    // Проверка правил
    FOR L_j := 1 TO GVL_CONSTANTS.C_MAX_RULES DO
        IF VI_Rule_Actions[L_j].Active AND VI_Rule_Actions[L_j].Target_ID = L_i THEN
            IF VI_Rule_Actions[L_j].Action_Type = E_Rule_Action_Type.ACTION_SET_LIGHTING_BASE THEN
                L_Rule_Light_Active := TRUE;
                L_Rule_Light_Val := REAL_TO_BYTE(VI_Rule_Actions[L_j].Value);
                L_Light_States[L_i] := (L_Rule_Light_Val > 0);
            ELSIF VI_Rule_Actions[L_j].Action_Type = E_Rule_Action_Type.ACTION_TOGGLE_LIGHTING AND VI_Rule_Actions[L_j].Triggered THEN
                L_Light_States[L_i] := NOT L_Light_States[L_i];
            END_IF;
        END_IF;
    END_FOR;

    // Приоритет 1: Физические выключатели (ТЗ 1.0)
    IF VI_Physical_Switches[L_i] AND NOT L_Prev_Switches[L_i] THEN
        L_Light_States[L_i] := NOT L_Light_States[L_i];
        L_Manual_Override[L_i] := TRUE; // Запоминаем ручное переопределение
    END_IF;
    L_Prev_Switches[L_i] := VI_Physical_Switches[L_i];

    // Приоритет 2: Датчики движения (ТЗ 2.0)
    // Защита от дребезга и удержание сигнала движения с помощью TOF
    L_Motion_Timers[L_i](IN := VI_Motion_Sensors[L_i], PT := T#5m, VI_System_Time_MS := VI_System_Time_MS);
    
    // Сброс ручного переопределения, когда комната становится пустой (задний фронт таймера движения)
    IF L_Prev_Motion_Q[L_i] AND NOT L_Motion_Timers[L_i].Q THEN
        L_Manual_Override[L_i] := FALSE;
    END_IF;
    L_Prev_Motion_Q[L_i] := L_Motion_Timers[L_i].Q;

    IF L_Motion_Timers[L_i].Q THEN
        IF NOT L_Manual_Override[L_i] THEN
            L_Light_States[L_i] := TRUE;
        END_IF;
    ELSE
        // Выключаем свет только если нет ручного переопределения
        IF NOT L_Manual_Override[L_i] THEN
            L_Light_States[L_i] := FALSE;
        END_IF;
    END_IF;

    // Приоритет 3: Симуляция (только в режиме Away)
    IF L_Effective_Scenario = E_SCENARIO_TYPE.SCENARIO_AWAY AND L_Effective_Simulation_Active THEN
        L_Light_States[L_i] := VI_Simulation_Lights[L_i];
    END_IF;

    // Приоритет 4: Ручное управление и правила
    IF VI_Manual_Light_Override[L_i] > 0 THEN
        VO_Lighting_Levels[L_i] := VI_Manual_Light_Override[L_i];
    ELSIF L_Rule_Light_Active THEN
        VO_Lighting_Levels[L_i] := L_Rule_Light_Val;
    ELSE
        VO_Lighting_Levels[L_i] := SEL(L_Light_States[L_i], 0, L_Base_Light);
    END_IF;
    
    // 5. Мокрые зоны
    IF VI_Wet_Zone_Map[L_i] AND L_Wet_Zone_Idx <= GVL_CONSTANTS.C_MAX_WET_ZONES THEN
        VO_Wet_Zone_Light_Active[L_Wet_Zone_Idx] := (VO_Lighting_Levels[L_i] > 10);
        L_Wet_Zone_Idx := L_Wet_Zone_Idx + 1;
    END_IF;
END_FOR;

// 3. Управление шторами
FOR L_i := 1 TO GVL_CONSTANTS.C_MAX_BLINDS DO
    L_Rule_Blinds_Active := FALSE;
    L_Rule_Blinds_Val := 0;
    
    // Проверка правил
    FOR L_j := 1 TO GVL_CONSTANTS.C_MAX_RULES DO
        IF VI_Rule_Actions[L_j].Active AND VI_Rule_Actions[L_j].Target_ID = L_i THEN
            IF VI_Rule_Actions[L_j].Action_Type = E_Rule_Action_Type.ACTION_SET_BLINDS THEN
                L_Rule_Blinds_Active := TRUE;
                L_Rule_Blinds_Val := REAL_TO_BYTE(VI_Rule_Actions[L_j].Value);
            END_IF;
        END_IF;
    END_FOR;

    // Приоритет 1: Ручное управление
    IF VI_Manual_Blinds_Override[L_i] > 0 THEN
        VO_Blinds_Positions[L_i] := VI_Manual_Blinds_Override[L_i];
    // Приоритет 2: Правила
    ELSIF L_Rule_Blinds_Active THEN
        VO_Blinds_Positions[L_i] := L_Rule_Blinds_Val;
    // Приоритет 3: Сценарий
    ELSE
        VO_Blinds_Positions[L_i] := L_Base_Blinds;
    END_IF;
END_FOR;

// ========================================
// Lighting V2 shadow execution (phase2)
// ========================================
fbLightingV2Staging(
    VI_Zone_ID := 1,
    VI_Enable := (VO_Lighting_Levels[1] > 0),
    VI_Brightness_Setpoint := BYTE_TO_REAL(VO_Lighting_Levels[1]),
    VI_Scene_ID := TO_INT(L_Effective_Scenario),
    VI_Manual_Override := (VI_Manual_Light_Override[1] > 0),
    VI_Transition_Time_MS := 5000,

    VI_Is_Active := (VO_Lighting_Levels[1] > 0),
    VI_Brightness_Actual := BYTE_TO_REAL(VO_Lighting_Levels[1]),
    VI_Motion_Active := VI_Motion_Sensors[1],
    VI_Ambient_Lux := 0.0,
    VI_Alarm_Active := GVL_STATE.G_Lighting_IO_Fault OR GVL_STATE.G_Lighting_Subsystem_Degraded,

    VO_Command_Shadow => L_Lighting_V2_Command_Shadow,
    VO_State_Shadow => L_Lighting_V2_State_Shadow
);

// ========================================
// Lighting V2 shadow validation
// ========================================
IF ABS(BYTE_TO_REAL(VO_Lighting_Levels[1]) - L_Lighting_V2_Command_Shadow.Brightness_Setpoint) > 0.1 THEN
    L_Lighting_V2_Shadow_Diff_Found := TRUE;
END_IF;
IF ABS(BYTE_TO_REAL(VO_Lighting_Levels[1]) - L_Lighting_V2_State_Shadow.Brightness_Actual) > 0.1 THEN
    L_Lighting_V2_Shadow_Diff_Found := TRUE;
END_IF;
IF VI_Motion_Sensors[1] <> L_Lighting_V2_State_Shadow.Motion_Active THEN
    L_Lighting_V2_Shadow_Diff_Found := TRUE;
END_IF;

// Guarded Lighting V2 enable
IF L_Lighting_V2_Switch_Enabled THEN
    IF NOT L_Lighting_V2_Shadow_Diff_Found THEN
        L_Lighting_V2_Path_Ready := TRUE;
        L_Lighting_Using_Legacy_Fallback := FALSE;
    ELSE
        L_Lighting_V2_Path_Ready := FALSE;
        L_Lighting_Using_Legacy_Fallback := TRUE;
    END_IF;
ELSE
    L_Lighting_V2_Path_Ready := FALSE;
    L_Lighting_Using_Legacy_Fallback := TRUE;
END_IF;



// ========================================
// Blinds V2 shadow execution (phase2)
// ========================================
fbBlindsV2Staging(
    VI_Blind_ID := 1,
    VI_Enable := TRUE,
    VI_Position_Setpoint := VO_Blinds_Positions[1],
    VI_Manual_Override := (VI_Manual_Blinds_Override[1] > 0),
    VI_Scenario_ID := TO_INT(L_Effective_Scenario),
    VI_Safety_Mode := FALSE,

    VI_Position_Actual := VO_Blinds_Positions[1],
    VI_Manual_Override_Active := (VI_Manual_Blinds_Override[1] > 0),
    VI_Is_Moving := FALSE,
    VI_Alarm_Active := GVL_STATE.G_Lighting_IO_Fault,

    VO_Command_Shadow => L_Blinds_V2_Command_Shadow,
    VO_State_Shadow => L_Blinds_V2_State_Shadow
);

// Blinds validation
IF VO_Blinds_Positions[1] <> L_Blinds_V2_Command_Shadow.Position_Setpoint THEN
    L_Blinds_V2_Shadow_Diff_Found := TRUE;
END_IF;
IF VO_Blinds_Positions[1] <> L_Blinds_V2_State_Shadow.Position_Actual THEN
    L_Blinds_V2_Shadow_Diff_Found := TRUE;
END_IF;


// Guarded Blinds V2 enable
IF L_Blinds_V2_Switch_Enabled THEN
    IF NOT L_Blinds_V2_Shadow_Diff_Found THEN
        L_Blinds_V2_Path_Ready := TRUE;
        L_Blinds_Using_Legacy_Fallback := FALSE;
    ELSE
        L_Blinds_V2_Path_Ready := FALSE;
        L_Blinds_Using_Legacy_Fallback := TRUE;
    END_IF;
ELSE
    L_Blinds_V2_Path_Ready := FALSE;
    L_Blinds_Using_Legacy_Fallback := TRUE;
END_IF;

END_FUNCTION_BLOCK

          
END_FUNCTION_BLOCK

FUNCTION_BLOCK FB_Maintenance_Access
  VAR_INPUT
    VI_System_Time : UDINT;
    VI_Activate : BOOL;
    VI_Duration : UDINT := 60;  (* мин *)
  END_VAR
  VAR_OUTPUT
    VO_Active : BOOL;
    VO_Time_Left : UDINT;
  END_VAR
  VAR
    L_Start_Time : UDINT;
    L_elapsed : UDINT;
  END_VAR

            IF VI_Activate AND NOT VO_Active THEN
    VO_Active := TRUE;
    L_Start_Time := VI_System_Time;
END_IF;

IF VO_Active THEN
    L_elapsed := (VI_System_Time - L_Start_Time) / 60000;
    IF L_elapsed >= VI_Duration THEN
        VO_Active := FALSE;
    ELSE
        VO_Time_Left := VI_Duration - L_elapsed;
    END_IF;
END_IF;

          
END_FUNCTION_BLOCK

FUNCTION_BLOCK FB_Manifold_Mixing_Valve_Controller
  VAR_INPUT
    VI_Setpoint : REAL;
    VI_Actual : REAL;
  END_VAR
  VAR_OUTPUT
    VO_Valve_Pos : REAL;  (* 0-100% *)
  END_VAR

            // ПИД-регулятор (упрощенно для примера)
VO_Valve_Pos := (VI_Setpoint - VI_Actual) * 10.0;
IF VO_Valve_Pos > 100.0 THEN VO_Valve_Pos := 100.0;
ELSIF VO_Valve_Pos < 0.0 THEN VO_Valve_Pos := 0.0;
END_IF;

          
END_FUNCTION_BLOCK

FUNCTION_BLOCK FB_Manifold_Pump_Controller
  VAR_INPUT
    VI_Enable_Request : BOOL;
    VI_System_Time : UDINT;
    VI_Stop_Ramp_MS : UDINT := 5000;
  END_VAR
  VAR_OUTPUT
    VO_Speed_Percent : BYTE;
    VO_Running : BOOL;
  END_VAR
  VAR
    L_Stop_Start_Time : UDINT;
    L_Stopping : BOOL;
    L_elapsed : UDINT;
  END_VAR

            IF VI_Enable_Request THEN
    VO_Speed_Percent := 100;
    VO_Running := TRUE;
    L_Stopping := FALSE;
ELSE
    IF VO_Running AND NOT L_Stopping THEN
        L_Stopping := TRUE;
        L_Stop_Start_Time := VI_System_Time;
    END_IF;
    
    IF L_Stopping THEN
        L_elapsed := VI_System_Time - L_Stop_Start_Time;
        IF L_elapsed < VI_Stop_Ramp_MS THEN
            // Исправлено: защита от отрицательного значения
            VO_Speed_Percent := REAL_TO_BYTE(100.0 * (1.0 - TO_REAL(L_elapsed) / TO_REAL(VI_Stop_Ramp_MS)));
        ELSE
            VO_Speed_Percent := 0;
            VO_Running := FALSE;
            L_Stopping := FALSE;
        END_IF;
    END_IF;
END_IF;

          
END_FUNCTION_BLOCK

FUNCTION_BLOCK FB_Manual_Valve_Control
  VAR_INPUT
    VI_System_Time : UDINT;
    VI_Open_Req : BOOL;
    VI_Duration : UDINT := 5;  (* мин *)
  END_VAR
  VAR_OUTPUT
    VO_Open_Cmd : BOOL;
    VO_Time_Left : UDINT;
  END_VAR
  VAR
    L_Start_Time : UDINT;
    L_Active : BOOL;
    L_elapsed : UDINT;
  END_VAR

            // Логика ручного управления клапаном с таймером автозакрытия
IF VI_Open_Req AND NOT L_Active THEN
    L_Active := TRUE;
    L_Start_Time := VI_System_Time;
    VO_Open_Cmd := TRUE;
END_IF;

IF L_Active THEN
    // Расчет оставшегося времени в минутах
    L_elapsed := (VI_System_Time - L_Start_Time) / 60000;
    IF L_elapsed >= VI_Duration THEN
        L_Active := FALSE;
        VO_Open_Cmd := FALSE;
    ELSE
        VO_Time_Left := VI_Duration - L_elapsed;
    END_IF;
ELSE
    VO_Time_Left := 0;
END_IF;

          
END_FUNCTION_BLOCK

FUNCTION_BLOCK FB_NVRAM_Manager
  VAR_INPUT
    VI_Command : BYTE;  (* 1=WRITE, 2=READ, 3=FORMAT *)
    VI_RecordIndex : INT;
    VI_DataPtr : POINTER TO BYTE;
    VI_DataSize : UDINT;  (* КРИТИЧНО: используем этот размер вместо SIZEOF *)
    VI_System_Time_MS : UDINT;
    VI_Operator_ID : STRING(10);
    VI_IsActivePLC : BOOL;
    VI_TwoPersonConfirmation : BOOL;
  END_VAR
  VAR_OUTPUT
    VO_Done : BOOL;
    VO_Error : UDINT;
    VO_ErrorID : UDINT;
    VO_ReadDataPtr : POINTER TO BYTE;
    VO_HMI_Status_Message : STRING(200);
  END_VAR
  VAR
    L_state : BYTE;
    L_step : UDINT;
    L_temp_buffer : ARRAY[1..132] OF BYTE;
    L_crc32 : FB_CRC32_Calculator;
    L_confirm_start_time : UDINT;
    L_cmd_copy : BYTE;
    L_prev_Command : BYTE;
    L_i : UDINT;
    L_current_time : UDINT;
    L_cmd_rising : BOOL;
    L_data_crc : DWORD;
    L_FileHandle : RTS_IEC_HANDLE;
    L_FileName : STRING := '/home/root/nvram_data.bin';
    L_FileResult : RTS_IEC_RESULT;
    L_BytesProcessed : UDINT;
    L_BackupIdx : INT := 1;  (* Для ротации *)
    L_Offset : DINT;
  END_VAR
  VAR CONSTANT
    C_MAGIC_NUMBER : UDINT := 16#534D5254;  (* "SMRT" *)
    C_STRUCT_VERSION : UINT := 21;  (* ТЗ v21.0 *)
    C_NVRAM_BASE_ADDR : UDINT := 16#20000;
    C_HEADER_SIZE : UDINT := 12;
    C_RECORD_SIZE : UDINT := 128;
    C_RECORD_TOTAL_SIZE : UDINT := 132;
    C_MAX_RECORDS : UDINT := 96;
    C_TWO_PERSON_TIMEOUT_MS : UDINT := 120000;
  END_VAR

            // Детекция фронта команды
L_cmd_rising := (VI_Command <> 0) AND (L_prev_Command = 0);
L_prev_Command := VI_Command;

IF L_cmd_rising THEN
    VO_Done := FALSE;
    VO_Error := FALSE;
    VO_ErrorID := 0;
    VO_HMI_Status_Message := '';
    
    // Валидация смещения
    IF VI_Offset >= C_MAX_NVRAM_SIZE THEN
        VO_Error := TRUE;
        VO_ErrorID := 16#1501;
        VO_HMI_Status_Message := 'NVRAM: Неверное смещение';
        VO_Done := TRUE;
        RETURN;
    END_IF;

    // Валидация указателя
    IF NOT __ISVALIDREF(VI_DataRef) THEN
        VO_Error := TRUE;
        VO_ErrorID := 16#150A;
        VO_HMI_Status_Message := 'NVRAM: Недействительная ссылка на данные';
        VO_Done := TRUE;
        RETURN;
    END_IF;

    IF (VI_Offset + VI_DataSize) > C_MAX_NVRAM_SIZE THEN
        VO_Error := TRUE;
        VO_ErrorID := 16#150B;
        VO_HMI_Status_Message := 'NVRAM: Размер данных превышает доступный объем';
        VO_Done := TRUE;
        RETURN;
    END_IF;

    IF VI_Command = 1 THEN // ЗАПИСЬ (WRITE)
        IF NOT VI_IsActivePLC THEN
            VO_Error := TRUE;
            VO_ErrorID := 16#1509;
            VO_HMI_Status_Message := 'NVRAM: Запись запрещена (STANDBY)';
        ELSE
            // Ограничение частоты записи (не чаще 1 раза в 60 секунд)
            IF F_TimeDiff(VI_System_Time_MS, L_Last_Write_Time_MS) < 60000 AND L_Last_Write_Time_MS <> 0 THEN
                VO_Error := TRUE;
                VO_ErrorID := 16#150C;
                VO_HMI_Status_Message := 'NVRAM: Превышена частота записи (лимит 1 раз в 60с)';
            ELSE
                // Проверка на изменение данных перед записью
                L_Data_Changed := FALSE;
                IF MEMCMP(ADR(GVL_Retain.G_NVRAM_Data[VI_Offset]), ADR(VI_DataRef), VI_DataSize) <> 0 THEN
                    L_Data_Changed := TRUE;
                END_IF;
                
                IF L_Data_Changed THEN
                    // Копируем данные используя MEMCPY
                    MEMCPY(ADR(GVL_Retain.G_NVRAM_Data[VI_Offset]), ADR(VI_DataRef), VI_DataSize);
                    L_Last_Write_Time_MS := VI_System_Time_MS;
                    VO_HMI_Status_Message := 'NVRAM: Данные успешно сохранены в RETAIN';
                ELSE
                    VO_HMI_Status_Message := 'NVRAM: Данные не изменились, запись пропущена';
                END_IF;
            END_IF;
        END_IF;
        VO_Done := TRUE;
        
    ELSIF VI_Command = 2 THEN // ЧТЕНИЕ (READ)
        // Копируем данные используя MEMCPY
        MEMCPY(ADR(VI_DataRef), ADR(GVL_Retain.G_NVRAM_Data[VI_Offset]), VI_DataSize);
        VO_ReadDataRef REF= VI_DataRef;
        VO_HMI_Status_Message := 'NVRAM: Данные успешно прочитаны из RETAIN';
        VO_Done := TRUE;
    END_IF;
END_IF;

IF VI_Command = 0 THEN
    VO_Done := FALSE;
END_IF;

          
END_FUNCTION_BLOCK

FUNCTION_BLOCK FB_Outdoor_Lighting_Controller
  VAR_INPUT
    VI_Ambient_Lux : REAL;
    VI_Motion : BOOL;
    VI_Security : BOOL;
  END_VAR
  VAR_OUTPUT
    VO_Light_On : BOOL;
  END_VAR

            IF VI_Security AND VI_Motion THEN
    VO_Light_On := TRUE; // Тревожное освещение
ELSIF VI_Ambient_Lux < 50.0 THEN
    VO_Light_On := TRUE; // Ночное освещение
ELSE
    VO_Light_On := FALSE;
END_IF;

          
END_FUNCTION_BLOCK

FUNCTION_BLOCK FB_PID_Controller
  VAR_INPUT
    VI_SetPoint : REAL;  (* Уставка *)
    VI_ProcessValue : REAL;  (* Текущее значение *)
    VI_Kp : REAL;  (* Коэффициент усиления *)
    VI_Tn : REAL;  (* Время интегрирования (сек) *)
    VI_Tv : REAL;  (* Время дифференцирования (сек) *)
    VI_Y_Min : REAL := 0;  (* Минимальный выход *)
    VI_Y_Max : REAL := 100;  (* Максимальный выход *)
    VI_Manual_Mode : BOOL;  (* Ручной режим *)
    VI_Manual_Value : REAL;  (* Значение в ручном режиме *)
    VI_Deadband : REAL := 0.1;  (* Мертвая зона *)
    VI_Cycle_Time_S : REAL := 0.01;  (* Время цикла задачи в секундах *)
    VI_Reset : BOOL;  (* Сброс интегральной составляющей *)
  END_VAR
  VAR_OUTPUT
    VO_Output : REAL;  (* Выход регулятора *)
    VO_Error : REAL;  (* Ошибка рассогласования *)
    VO_Limiting : BOOL;  (* Флаг ограничения выхода (Anti-windup) *)
  END_VAR
  VAR
    L_Integral_Sum : REAL;  (* Интегральная сумма *)
    L_Prev_Error : REAL;  (* Предыдущая ошибка *)
    L_Derivative : REAL;  (* Дифференциальная составляющая *)
    L_Output_Raw : REAL;  (* Сырой выход до ограничения *)
  END_VAR

            // Расчет ошибки
VO_Error := VI_SetPoint - VI_ProcessValue;

// Проверка мертвой зоны
IF ABS(VO_Error) < VI_Deadband THEN
    VO_Error := 0.0;
END_IF;

IF VI_Reset THEN
    L_Integral_Sum := 0.0;
    L_Prev_Error := 0.0;
    VO_Output := 0.0;
    RETURN;
END_IF;

IF VI_Manual_Mode THEN
    VO_Output := VI_Manual_Value;
    // Безударный переход: при выходе из ручного режима выход должен остаться прежним.
    // Так как Выход = P + I + D, то I = Выход - P - D.
    // Для простоты D при переходе обнуляем (или игнорируем), тогда I = Выход - P.
    L_Integral_Sum := VO_Output - (VI_Kp * VO_Error);
    L_Prev_Error := VO_Error;
    RETURN;
END_IF;

// Пропорциональная составляющая
L_Output_Raw := VI_Kp * VO_Error;

// Интегральная составляющая (Метод трапеций)
IF VI_Tn > 0.0 THEN
    // Anti-windup: не накапливаем интеграл, если выход уже на пределе и ошибка того же знака
    IF NOT VO_Limiting OR (VO_Error > 0.0 AND L_Output_Raw < VI_Y_Max) OR (VO_Error < 0.0 AND L_Output_Raw > VI_Y_Min) THEN
        L_Integral_Sum := L_Integral_Sum + (VI_Kp / VI_Tn) * VO_Error * VI_Cycle_Time_S;
    END_IF;
    L_Output_Raw := L_Output_Raw + L_Integral_Sum;
END_IF;

// Дифференциальная составляющая
IF VI_Tv > 0.0 THEN
    L_Derivative := (VO_Error - L_Prev_Error) / VI_Cycle_Time_S;
    L_Output_Raw := L_Output_Raw + VI_Kp * VI_Tv * L_Derivative;
END_IF;

L_Prev_Error := VO_Error;

// Ограничение выхода
IF L_Output_Raw > VI_Y_Max THEN
    VO_Output := VI_Y_Max;
    VO_Limiting := TRUE;
ELSIF L_Output_Raw < VI_Y_Min THEN
    VO_Output := VI_Y_Min;
    VO_Limiting := TRUE;
ELSE
    VO_Output := L_Output_Raw;
    VO_Limiting := FALSE;
END_IF;

          
END_FUNCTION_BLOCK

FUNCTION_BLOCK FB_PLC_Heartbeat
  VAR_INPUT
    VI_Local_ID : BYTE;
    VI_System_Time : UDINT;
    VI_Remote_Pulse : BOOL;
    VI_Remote_Is_Active : BOOL;  (* ТЗ 8.3: Уровень 2 - проверка роли партнера *)
    VI_Gateway_Ping_OK : BOOL;  (* ТЗ 8.3: Уровень 3 - пинг шлюза *)
  END_VAR
  VAR_OUTPUT
    VO_Is_Active : BOOL;
    VO_RTT_MS : UDINT;
    VO_Loss_Count : UDINT;  (* ТЗ 8.4: Статистика потерь *)
    VO_Max_RTT : UDINT;  (* ТЗ 8.4: Макс. задержка *)
  END_VAR
  VAR
    L_Last_Pulse : BOOL;
    L_Last_Pulse_Time : UDINT;
    L_Timeout : UDINT := 500;  (* ТЗ 8.1: 500 мс *)
    L_Pulse_Send_Time : UDINT;
    L_Loss_Timer : TON;
  END_VAR

            // 1. Мониторинг пульса и RTT (ТЗ 8.4)
IF VI_Remote_Pulse <> L_Last_Pulse THEN
    VO_RTT_MS := VI_System_Time - L_Last_Pulse_Time;
    IF VO_RTT_MS > VO_Max_RTT THEN VO_Max_RTT := VO_RTT_MS; END_IF;
    L_Last_Pulse := VI_Remote_Pulse;
    L_Last_Pulse_Time := VI_System_Time;
END_IF;

L_Loss_Timer(IN := (VI_System_Time - L_Last_Pulse_Time) > L_Timeout, PT := T#1s);
IF L_Loss_Timer.Q THEN 
    VO_Loss_Count := VO_Loss_Count + 1; 
    L_Loss_Timer(IN := FALSE); 
END_IF;

// 2. Логика активности и защита от раскола мозга (ТЗ 8.3)
// Уровень 1: Тайм-аут пульса
IF (VI_System_Time - L_Last_Pulse_Time) < L_Timeout THEN
    // Уровень 2: Если партнер заявляет, что он активен, и у него приоритет (ID=1)
    IF VI_Remote_Is_Active AND VI_Local_ID = 2 THEN
        VO_Is_Active := FALSE;
    ELSE
        // Приоритет у ПЛК A (ID=1)
        VO_Is_Active := (VI_Local_ID = 1);
    END_IF;
ELSE
    // Уровень 3: Если связи нет, проверяем доступность шлюза
    VO_Is_Active := VI_Gateway_Ping_OK OR (VI_Local_ID = 1);
END_IF;

          
END_FUNCTION_BLOCK

FUNCTION_BLOCK FB_Pre_Departure_Heating
  VAR_INPUT
    VI_Departure_Time : UDINT;
    VI_System_Time : UDINT;
    VI_Selected : ARRAY[1..16] OF BOOL;
  END_VAR
  VAR_OUTPUT
    VO_Heating_Active : BOOL;
    VO_Setpoints : ARRAY[1..16] OF REAL;
  END_VAR
  VAR
    L_i : INT;
  END_VAR

            // Запуск за 3 часа (10800000 мс)
IF (VI_Departure_Time - VI_System_Time) < 10800000 THEN
    VO_Heating_Active := TRUE;
    FOR L_i := 1 TO 16 DO
        IF VI_Selected[L_i] THEN VO_Setpoints[L_i] := 22.0; END_IF;
    END_FOR;
ELSE
    VO_Heating_Active := FALSE;
END_IF;

          
END_FUNCTION_BLOCK

FUNCTION_BLOCK FB_Presence_Playback
  VAR_INPUT
    VI_Mode_Record : BOOL;  (* TRUE - записываем, FALSE - воспроизводим *)
    VI_Light_Inputs : ARRAY[1..16] OF BOOL;
    VI_Time_Index : UDINT;  (* Индекс времени в рамках недели (мс) *)
  END_VAR
  VAR_OUTPUT
    VO_Light_Outputs : ARRAY[1..16] OF BOOL;
  END_VAR
  VAR
    L_History : ARRAY[0..1007] OF WORD;  (* 168 часов * 6 записей в час = 1008 записей (битовая маска 16 ламп) *)
    L_Current_Slot : UDINT;
    L_i : INT;
  END_VAR

            L_Current_Slot := (VI_Time_Index / 600000) MOD 1008; // Слот каждые 10 минут

IF VI_Mode_Record THEN
    // Запись текущего состояния в слот
    L_History[L_Current_Slot] := 0;
    FOR L_i := 1 TO 16 DO
        IF VI_Light_Inputs[L_i] THEN
            L_History[L_Current_Slot] := L_History[L_Current_Slot] OR SHL(WORD#1, L_i-1);
        END_IF;
    END_FOR;
ELSE
    // Воспроизведение из слота
    FOR L_i := 1 TO 16 DO
        VO_Light_Outputs[L_i] := (L_History[L_Current_Slot] AND SHL(WORD#1, L_i-1)) <> 0;
    END_FOR;
END_IF;

          
END_FUNCTION_BLOCK

FUNCTION_BLOCK FB_Presence_Simulator
  VAR_INPUT
    VI_Enabled : BOOL;
    VI_Intensity : REAL;
    VI_System_Time : UDINT;
    VI_Use_Playback : BOOL;  (* Новый режим воспроизведения *)
  END_VAR
  VAR_OUTPUT
    VO_Light_States : ARRAY[1..16] OF BOOL;
  END_VAR
  VAR
    fbPlayback : FB_Presence_Playback;
  END_VAR

            IF VI_Enabled THEN
    IF VI_Use_Playback THEN
        fbPlayback(VI_Mode_Record := FALSE, VI_Time_Index := VI_System_Time MOD 604800000, VO_Light_Outputs => VO_Light_States);
    ELSE
        // Старая логика случайной симуляции
        VO_Light_States[1] := (VI_System_Time MOD 100000 > 50000);
    END_IF;
END_IF;

          
END_FUNCTION_BLOCK

FUNCTION_BLOCK FB_Random_Generator
  VAR
    L_seed : UDINT := 1;
  END_VAR
  VAR CONSTANT
    C_LCG_MULTIPLIER : UDINT := 1664525;
    C_LCG_INCREMENT : UDINT := 1013904223;
    C_LCG_MODULUS : LREAL := 4294967296;
  END_VAR

            
          

METHOD Random_Int_Range : UDINT
  VAR_INPUT
    VI_min : UDINT;
    VI_max : UDINT;
  END_VAR
  VAR
    L_range : UDINT;
    L_rand_factor : LREAL;
  END_VAR
                  L_seed := (C_LCG_MULTIPLIER * L_seed) + C_LCG_INCREMENT;

IF VI_max > VI_min THEN
        L_range := VI_max - VI_min;
        // Используем LREAL для точности и исключения выхода за границу
        L_rand_factor := TO_LREAL(L_seed) / C_LCG_MODULUS;
        Random_Int_Range := VI_min + TO_UDINT(L_rand_factor * TO_LREAL(L_range + 1));
        
        // Финальная защита от переполнения
        IF Random_Int_Range > VI_max THEN
            Random_Int_Range := VI_max;
        END_IF;
    ELSE
        Random_Int_Range := VI_min;
    END_IF;
                
END_METHOD
END_FUNCTION_BLOCK

FUNCTION_BLOCK FB_Scenario_Manager
  VAR_INPUT
    VI_System_Time_MS : UDINT;
    VI_Activate_Request : E_SCENARIO_TYPE;
    VI_IsActivePLC : BOOL;
  END_VAR
  VAR_OUTPUT
    VO_Current_Scenario : E_SCENARIO_TYPE;
    VO_Status_Msg : STRING(200);
  END_VAR

            IF NOT VI_IsActivePLC THEN
    RETURN;
END_IF;

CASE VI_System_Mode OF
    E_System_Operating_Mode.MODE_SAFE_STOP,
    E_System_Operating_Mode.MODE_FREEZE_PROTECTION:
        IF VO_Current_Scenario <> E_SCENARIO_TYPE.SCENARIO_NONE THEN
            VO_Current_Scenario := E_SCENARIO_TYPE.SCENARIO_NONE;
            VO_Status_Msg := 'Сценарии принудительно отключены режимом безопасности';
        END_IF;
        RETURN;

    E_System_Operating_Mode.MODE_DEGRADED:
        VO_Status_Msg := 'Смена сценариев заблокирована: деградированный режим';
        RETURN;
END_CASE;

IF VI_Activate_Request <> VO_Current_Scenario THEN
    // Проверка минимального времени работы сценария
    IF F_TimeDiff(VI_System_Time_MS, L_Last_Scenario_Time) >= 60000 OR VO_Current_Scenario = E_SCENARIO_TYPE.SCENARIO_NONE THEN
        // Логика переключения сценариев
        VO_Current_Scenario := VI_Activate_Request;
        L_Last_Scenario_Time := VI_System_Time_MS;
        
        CASE VO_Current_Scenario OF
        E_SCENARIO_TYPE.SCENARIO_NONE:
            VO_Status_Msg := 'Сценарии отключены';
        E_SCENARIO_TYPE.SCENARIO_AWAY:
            VO_Status_Msg := 'Активирован сценарий: Вне дома (Охрана + Энергосбережение)';
        E_SCENARIO_TYPE.SCENARIO_SLEEP:
            VO_Status_Msg := 'Активирован сценарий: Сон (Ночное освещение + Климат)';
        E_SCENARIO_TYPE.SCENARIO_PRESENCE:
            VO_Status_Msg := 'Активирован сценарий: Имитация присутствия';
        END_CASE;
    END_IF;
END_IF;

          
END_FUNCTION_BLOCK

FUNCTION_BLOCK FB_Scenario_Transition_Controller
  VAR_INPUT
    VI_System_Time : UDINT;
    VI_Start_Time : UDINT;
    VI_Min_Dur : UDINT := 300000;  (* 5 мин *)
  END_VAR
  VAR_OUTPUT
    VO_Allowed : BOOL;
  END_VAR

            VO_Allowed := (VI_System_Time - VI_Start_Time) >= VI_Min_Dur;

          
END_FUNCTION_BLOCK

FUNCTION_BLOCK FB_Security_Alarm
  VAR_INPUT
    VI_IsActivePLC : BOOL;
    VI_Assigned_DoorWindow_Open : ARRAY[1..20] OF BOOL;
    VI_Assigned_GlassBreak : ARRAY[1..12] OF BOOL;
  END_VAR
  VAR_OUTPUT
    VO_Alarm_Active : BOOL;
    VO_Status_Msg : STRING(200);
  END_VAR

            VO_Alarm_Active := CheckPerimeter();

IF VO_Alarm_Active THEN
    VO_Status_Msg := 'ТРЕВОГА: НАРУШЕН ПЕРИМЕТР';
ELSE
    VO_Status_Msg := 'Периметр в норме';
END_IF;


          

METHOD CheckPerimeter : BOOL
  VAR
    L_i : INT;
  END_VAR
                  CheckPerimeter := FALSE;
// Проверка окон
FOR L_i := 1 TO 20 DO
    IF VI_Assigned_DoorWindow_Open[L_i] THEN
        CheckPerimeter := TRUE;
        RETURN;
    END_IF;
END_FOR;
// Проверка стекол
FOR L_i := 1 TO 12 DO
    IF VI_Assigned_GlassBreak[L_i] THEN
        CheckPerimeter := TRUE;
        RETURN;
    END_IF;
END_FOR;
                
END_METHOD
END_FUNCTION_BLOCK

FUNCTION_BLOCK FB_Security_System
  VAR_INPUT
    VI_System_Time : UDINT;
    VI_Sensors_Open : ARRAY[1..15] OF BOOL;
    VI_Sensors_Glass : ARRAY[1..15] OF BOOL;
    VI_Grouped_2F : BOOL;
    VI_PIN_Code : STRING(4);
    VI_Arm_Request : BOOL;
  END_VAR
  VAR_OUTPUT
    VO_Alarm_Active : BOOL;
    VO_Alarm_Level : E_ALERT_PRIORITY;
    VO_Status : BYTE;  (* 0-Disarmed, 1-Arming, 2-Armed, 3-Alarm *)
  END_VAR
  VAR
    L_Last_Trigger_Time : UDINT;
    L_Trigger_Count : INT;
    L_i : INT;
  END_VAR

            L_Trigger_Count := 0;
FOR L_i := 1 TO 15 DO
    IF VI_Sensors_Open[L_i] OR VI_Sensors_Glass[L_i] THEN
        L_Trigger_Count := L_Trigger_Count + 1;
    END_IF;
END_FOR;
IF VI_Grouped_2F THEN L_Trigger_Count := L_Trigger_Count + 1; END_IF;

// Логика п. 3.3: Комбинированные события (>=2 датчиков за 10 сек)
IF L_Trigger_Count >= 2 THEN
    IF (VI_System_Time - L_Last_Trigger_Time) < 10000 THEN
        VO_Alarm_Level := E_ALERT_PRIORITY.ALERT_PRIORITY_CRITICAL;
        VO_Alarm_Active := TRUE;
    END_IF;
    L_Last_Trigger_Time := VI_System_Time;
END_IF;

          
END_FUNCTION_BLOCK

FUNCTION_BLOCK FB_Security_System_Manager
  VAR_INPUT
    VI_System_Time_MS : UDINT;
    VI_IsActivePLC : BOOL;
    VI_Opening_Sensors : ARRAY[1..15] OF BOOL;
    VI_GlassBreak_Sensors : ARRAY[1..15] OF BOOL;
    VI_PIN_Input : STRING(4);
    VI_PIN_Submit : BOOL;
    VI_Config : ST_Security_Config;
    VI_Outdoor_Lux : REAL;
    VI_Motion_Corridor : BOOL;
    VI_Acknowledge_Open_Windows : BOOL;  (* ТЗ 3.8 *)
    VI_Group_2F_Open : BOOL;  (* ТЗ 3.1 (7 окон -> 1 канал) *)
    VI_Group_2F_Glass : BOOL;  (* ТЗ 3.2 *)
  END_VAR
  VAR_OUTPUT
    VO_Armed : BOOL;
    VO_Alarm_Active : BOOL;
    VO_Entry_Delay_Active : BOOL;
    VO_Time_To_Alarm_S : UINT;
    VO_Away_Level : BYTE;  (* 1-Short, 2-Medium, 3-Long *)
    VO_Light_Corridor : BOOL;
    VO_Light_Stairs_Dim : BYTE;
    VO_Status_Msg : STRING(200);
    VO_Long_Away_Req : BOOL;  (* ТЗ 3.6: При тревоге -> долгосрочный отъезд *)
  END_VAR
  VAR
    L_State : BYTE;  (* 0-Disarmed, 1-Armed, 2-EntryDelay, 3-Alarm, 4-ConfirmWait *)
    L_Attempts : UINT;
    L_Entry_Start_Time : UDINT;
    L_Away_Start_Time : UDINT;
    L_Confirm_Start_Time : UDINT;
    L_Last_Trigger_Time : UDINT;
    L_i : INT;
    L_Any_Sensor_Open : BOOL;
    L_Any_Glass_Broken : BOOL;
    L_Trigger_Count : UINT;  (* ТЗ 3.3: Комбинированные события (>=2 за 10с) *)
    L_Trigger_Timer : TON;
    L_Last_Sensors : ARRAY[1..32] OF BOOL;
    L_Glass_Threshold_Multiplier : REAL := 1;  (* ТЗ 3.8: Снижение порога *)
  END_VAR

            IF NOT VI_IsActivePLC THEN RETURN; END_IF;

// 1. Проверка PIN-кода или RFID-метки через менеджер кодов
fbAccessCode(
    VI_System_Time_MS := VI_System_Time_MS,
    VI_IsActivePLC := VI_IsActivePLC,
    VI_Code_To_Check := VI_PIN_Code,
    VI_RFID_To_Check := VI_RFID_Tag,
    VO_Code_Valid => L_Valid_PIN
);

// 2. Логика постановки на охрану (с задержкой на выход)
L_Auto_Arm_Trigger := FALSE;
IF VI_Config.auto_arm_enabled THEN
    IF VI_Current_TOD >= UDINT_TO_TOD(VI_Config.auto_arm_time_ms) THEN
        L_Auto_Arm_Trigger := TRUE;
    END_IF;
END_IF;
R_Trig_Auto_Arm(CLK := L_Auto_Arm_Trigger);

IF ((VI_Arm_Request AND L_Valid_PIN) OR R_Trig_Auto_Arm.Q) AND NOT VO_Armed AND NOT L_Arming_In_Progress THEN
    // Проверка, что все двери/окна закрыты перед постановкой (с учетом байпаса)
    L_Any_Sensor_Active := FALSE;
    FOR L_i := 1 TO GVL_CONSTANTS.C_MAX_DOOR_SENSORS DO IF VI_Door_Sensors[L_i] AND NOT VI_Bypass_Doors[L_i] THEN L_Any_Sensor_Active := TRUE; END_IF; END_FOR;
    FOR L_i := 1 TO GVL_CONSTANTS.C_MAX_CLIMATE_ZONES DO IF VI_Window_Sensors[L_i] AND NOT VI_Bypass_Windows[L_i] THEN L_Any_Sensor_Active := TRUE; END_IF; END_FOR;
    
    IF NOT L_Any_Sensor_Active THEN
        L_Arming_In_Progress := TRUE;
        VO_Status_Msg := 'Постановка на охрану. Покиньте помещение.';
    ELSE
        VO_Status_Msg := 'Ошибка постановки: Открыты двери или окна';
    END_IF;
END_IF;

L_Arm_Delay_Timer(IN := L_Arming_In_Progress, PT := TO_TIME(VI_Config.exit_delay_seconds * 1000), VI_System_Time_MS := VI_System_Time_MS);
IF L_Arm_Delay_Timer.Q THEN
    L_Arming_In_Progress := FALSE;
    VO_Armed := TRUE;
    VO_Status_Msg := 'Система под охраной';
END_IF;

// 3. Логика снятия с охраны с 2FA
IF VI_Disarm_Request AND L_Valid_PIN AND VO_Armed THEN
    IF VI_Config.enable_2fa THEN
        L_Disarm_Pending := TRUE;
        L_2FA_Required := TRUE;
        VO_Status_Msg := 'Ожидание 2FA для снятия с охраны';
    ELSE
        // Снятие без 2FA
        VO_Armed := FALSE;
        VO_Alarm_Active := FALSE;
        VO_Siren_Active := FALSE;
        L_Arming_In_Progress := FALSE;
        VO_Status_Msg := 'Система снята с охраны';
    END_IF;
END_IF;

fbTwoFactor(
    VI_System_Time_MS := VI_System_Time_MS,
    VI_Start_Auth := L_2FA_Required,
    VI_Method := E_TwoFactor_Method.TF_METHOD_TOTP, // Для примера
    VI_User_Code := VI_2FA_Code, // Используем отдельный вход для 2FA кода
    VI_Reset_Success := L_Reset_2FA
);

VO_Send_Code_Req := fbTwoFactor.VO_Send_Code_Req;
VO_Code_To_Send := fbTwoFactor.VO_Code_To_Send;

IF L_Disarm_Pending AND fbTwoFactor.VO_State.Is_Success THEN
    VO_Armed := FALSE;
    VO_Alarm_Active := FALSE;
    VO_Siren_Active := FALSE;
    L_Arming_In_Progress := FALSE;
    L_Disarm_Pending := FALSE;
    L_2FA_Required := FALSE;
    L_Reset_2FA := TRUE;
    VO_Status_Msg := 'Система снята с охраны';
ELSIF L_Disarm_Pending AND fbTwoFactor.VO_State.Is_Locked THEN
    L_Disarm_Pending := FALSE;
    L_2FA_Required := FALSE;
    L_Reset_2FA := FALSE;
    VO_Status_Msg := 'Ошибка 2FA: Превышено количество попыток';
ELSE
    L_Reset_2FA := FALSE;
END_IF;

// 4. Логика тревоги (с задержкой на вход)
IF VO_Armed THEN
    L_Any_Sensor_Active := FALSE;
    FOR L_i := 1 TO GVL_CONSTANTS.C_MAX_CLIMATE_ZONES DO IF VI_Motion_Sensors[L_i] AND NOT VI_Bypass_Motion[L_i] THEN L_Any_Sensor_Active := TRUE; END_IF; END_FOR;
    FOR L_i := 1 TO GVL_CONSTANTS.C_MAX_DOOR_SENSORS DO IF VI_Door_Sensors[L_i] AND NOT VI_Bypass_Doors[L_i] THEN L_Any_Sensor_Active := TRUE; END_IF; END_FOR;
    FOR L_i := 1 TO GVL_CONSTANTS.C_MAX_CLIMATE_ZONES DO IF VI_Window_Sensors[L_i] AND NOT VI_Bypass_Windows[L_i] THEN L_Any_Sensor_Active := TRUE; END_IF; END_FOR;
    
    // Защелкиваем факт нарушения периметра, чтобы кратковременное срабатывание датчика не сбрасывало таймер
    IF L_Any_Sensor_Active THEN
        L_Alarm_Delay_Timer.IN := TRUE;
    END_IF;
    
    L_Alarm_Delay_Timer(PT := TO_TIME(VI_Config.entry_delay_seconds * 1000), VI_System_Time_MS := VI_System_Time_MS);
    
    IF L_Alarm_Delay_Timer.Q THEN
        VO_Alarm_Active := TRUE;
        VO_Siren_Active := TRUE;
        VO_Status_Msg := 'ТРЕВОГА! Нарушение периметра';
    ELSIF L_Alarm_Delay_Timer.IN THEN
        VO_Status_Msg := 'Внимание! Введите PIN-код для отмены тревоги';
    END_IF;
ELSE
    L_Alarm_Delay_Timer(IN := FALSE, PT := T#0s, VI_System_Time_MS := VI_System_Time_MS); // Сброс таймера при снятии с охраны
END_IF;

          
END_FUNCTION_BLOCK

FUNCTION_BLOCK FB_Sensor_Calibration_Processor
  VAR_INPUT
    VI_Raw_Value : REAL;
    VI_Calib_Record : ST_Sensor_Calibration_Record;
  END_VAR
  VAR_OUTPUT
    VO_Calibrated_Value : REAL;
  END_VAR

            // Формула: (Сырое значение * Множитель) + Смещение
VO_Calibrated_Value := (VI_Raw_Value * VI_Calib_Record.multiplier) + VI_Calib_Record.offset;

          
END_FUNCTION_BLOCK

FUNCTION_BLOCK FB_Sensor_Distribution
  VAR_INPUT
    VI_Local_PLC_ID : BYTE;  (* 1=A, 2=B *)
    VI_Raw_Sensors : ARRAY[1..20] OF BOOL;
  END_VAR
  VAR_OUTPUT
    VO_Assigned_Sensors : ARRAY[1..20] OF BOOL;
  END_VAR
  VAR
    L_i : INT;
  END_VAR

            FOR L_i := 1 TO 20 DO
    // ПЛК A берет четные, ПЛК B - нечетные
    IF (VI_Local_PLC_ID = 1 AND (L_i MOD 2 = 0)) OR
       (VI_Local_PLC_ID = 2 AND (L_i MOD 2 <> 0)) THEN
        VO_Assigned_Sensors[L_i] := VI_Raw_Sensors[L_i];
    END_IF;
END_FOR;

          
END_FUNCTION_BLOCK

FUNCTION_BLOCK FB_Simulation_Manager
  VAR_INPUT
    VI_System_Time_MS : UDINT;
    VI_Enabled : BOOL;
    VI_Intensity : REAL;  (* 0.2-0.3 *)
  END_VAR
  VAR_OUTPUT
    VO_Light_States : ARRAY[1..16] OF BOOL;
    VO_Socket_States : ARRAY[1..12] OF BOOL;
  END_VAR
  VAR
    L_Rand : FB_Random_Generator;
    L_Last_Event_Time : UDINT;
    L_Event_Duration : UDINT;
    L_Active : BOOL;
    L_i : INT;
    L_Current_TOD : TOD;
    L_In_Window : BOOL;
  END_VAR

            IF VI_Scenario = E_SCENARIO_TYPE.SCENARIO_AWAY AND VI_Config.Presence_Simulation_Enabled THEN
    VO_Sim_Active := TRUE;
    
    // Переключаем свет каждые 30 минут
    IF F_TimeDiff(VI_System_Time_MS, L_Last_Toggle) >= (GVL_CONSTANTS.C_MS_IN_MINUTE * 30) THEN
        L_Last_Toggle := VI_System_Time_MS;
        
        FOR L_i := 1 TO GVL_CONSTANTS.C_MAX_LIGHTING_ZONES DO
            L_Rand_Val := L_Random.Random_Int_Range(VI_min := 0, VI_max := 100);
            VO_Sim_Lights[L_i] := (L_Rand_Val > 80); // 20% шанс включения
        END_FOR;
    END_IF;
ELSE
    VO_Sim_Active := FALSE;
    FOR L_i := 1 TO GVL_CONSTANTS.C_MAX_LIGHTING_ZONES DO VO_Sim_Lights[L_i] := FALSE; END_FOR;
END_IF;

// Симуляция аварий в тестовом режиме
IF L_Test_Mode THEN
    // Генерация случайных протечек (очень редко)
    L_Rand_Val := L_Random.Random_Int_Range(VI_min := 0, VI_max := 100000);
    IF L_Rand_Val = 42 THEN
        VO_Sim_Water_Leak[1] := TRUE;
    END_IF;
    
    // Симуляция утечки газа
    L_Rand_Val := L_Random.Random_Int_Range(VI_min := 0, VI_max := 100000);
    IF L_Rand_Val = 77 THEN
        VO_Sim_Gas_Leak[1] := 15.0; // 15% LEL
    END_IF;
ELSE
    FOR L_i := 1 TO GVL_CONSTANTS.C_MAX_FLOOD_SENSORS DO VO_Sim_Water_Leak[L_i] := FALSE; END_FOR;
    FOR L_i := 1 TO GVL_CONSTANTS.C_MAX_METHANE_SENSORS DO VO_Sim_Gas_Leak[L_i] := 0.0; END_FOR;
END_IF;

          
END_FUNCTION_BLOCK

FUNCTION_BLOCK FB_Smoke_Detector
  VAR_INPUT
    VI_Sensors : ARRAY[1..6] OF BOOL;
    VI_System_Time : UDINT;
  END_VAR
  VAR_OUTPUT
    VO_Fire_Alarm : BOOL;
  END_VAR
  VAR
    L_Verify_Start : ARRAY[1..6] OF UDINT;
    L_Verifying : ARRAY[1..6] OF BOOL;
    L_i : INT;
  END_VAR

            FOR L_i := 1 TO 6 DO
    IF VI_Sensors[L_i] THEN
        IF NOT L_Verifying[L_i] THEN
            L_Verifying[L_i] := TRUE;
            L_Verify_Start[L_i] := VI_System_Time;
        ELSIF (VI_System_Time - L_Verify_Start[L_i]) > 30000 THEN
            VO_Fire_Alarm := TRUE;
        END_IF;
    ELSE
        L_Verifying[L_i] := FALSE;
    END_IF;
END_FOR;

          
END_FUNCTION_BLOCK

FUNCTION_BLOCK FB_SMS_Notification
  VAR_INPUT
    VI_Send_Request : BOOL;
    VI_Phone : STRING(15);
    VI_Text : STRING(160);
  END_VAR
  VAR_OUTPUT
    VO_Done : BOOL;
    VO_Error : BOOL;
  END_VAR
  VAR
    L_State : INT;
    L_Timer : TON;
    L_AT_Command : STRING(255);
  END_VAR

            CASE L_State OF
    0: // Ожидание запроса
        IF VI_Send_Request THEN
            VO_Done := FALSE;
            VO_Error := FALSE;
            L_State := 1;
        END_IF;
        
    1: // Отправка AT+CMGF=1 (Установка текстового режима)
        L_AT_Command := 'AT+CMGF=1$R';
        L_State := 2;
        L_Timer(IN := TRUE, PT := T#500ms);
        
    2: // Ожидание ответа OK и отправка номера
        L_Timer(IN := TRUE);
        IF L_Timer.Q THEN
            L_Timer(IN := FALSE);
            L_AT_Command := CONCAT('AT+CMGS="', CONCAT(VI_Phone, '"$R'));
            L_State := 3;
            L_Timer(IN := TRUE, PT := T#500ms);
        END_IF;
        
    3: // Отправка текста сообщения и символа Ctrl+Z (ASCII 26)
        L_Timer(IN := TRUE);
        IF L_Timer.Q THEN
            L_Timer(IN := FALSE);
            L_AT_Command := CONCAT(VI_Text, '$1A'); // $1A - это Ctrl+Z в CODESYS
            L_State := 4;
            L_Timer(IN := TRUE, PT := T#2s);
        END_IF;
        
    4: // Завершение
        L_Timer(IN := TRUE);
        IF L_Timer.Q THEN
            L_Timer(IN := FALSE);
            VO_Done := TRUE;
            L_State := 0;
        END_IF;
END_CASE;

          
END_FUNCTION_BLOCK

FUNCTION_BLOCK FB_State_Manager
  VAR_INPUT
    VI_System_Time_MS : UDINT;
    VI_Command : BYTE;  (* 1-Save, 2-Restore *)
    VI_Heating_Config : ST_Heating_Config;
  END_VAR
  VAR_OUTPUT
    VO_Heating_Config : ST_Heating_Config;
    VO_Done : BOOL;
  END_VAR
  VAR
    L_Saved_Heating : ST_Heating_Config;
    L_Restore_Start_Time : UDINT;
    L_Restoring : BOOL;
  END_VAR

            VO_System_OK := FALSE;
VO_System_Warning := FALSE;
VO_System_Critical := FALSE;
VO_Status_Msg := '';
VO_System_Mode := E_System_Operating_Mode.MODE_NORMAL;

CASE VI_System_Severity OF
    E_System_Severity.SEV_NORMAL:
        VO_System_OK := TRUE;
        VO_Status_Msg := 'Система в норме';
        VO_System_Mode := E_System_Operating_Mode.MODE_NORMAL;

    E_System_Severity.SEV_WARNING:
        VO_System_Warning := TRUE;
        VO_System_Mode := E_System_Operating_Mode.MODE_DEGRADED;
        CASE VI_Root_Cause OF
            E_System_Root_Cause.ROOT_WATER_LEAK:
                VO_Status_Msg := 'Предупреждение: протечка воды';
            E_System_Root_Cause.ROOT_CO_WARNING:
                VO_Status_Msg := 'Предупреждение: повышенный CO';
            ELSE
                VO_Status_Msg := 'Предупреждение системы';
        END_CASE;

    E_System_Severity.SEV_DEGRADED:
        VO_System_Warning := TRUE;
        VO_System_Mode := E_System_Operating_Mode.MODE_DEGRADED;
        CASE VI_Root_Cause OF
            E_System_Root_Cause.ROOT_SENSOR_FAULT:
                VO_Status_Msg := 'Деградация: ошибка датчика';
            E_System_Root_Cause.ROOT_IO_OFFLINE:
                VO_Status_Msg := 'Деградация: модуль IO недоступен';
            E_System_Root_Cause.ROOT_COMM_FAULT:
                VO_Status_Msg := 'Деградация: ошибка связи';
            E_System_Root_Cause.ROOT_WATCHDOG_FAULT:
                VO_Status_Msg := 'Деградация: watchdog fault';
            E_System_Root_Cause.ROOT_SUBSYSTEM_FAULT:
                VO_Status_Msg := 'Деградация: ошибка подсистемы';
            ELSE
                VO_Status_Msg := 'Деградация системы';
        END_CASE;

    E_System_Severity.SEV_CRITICAL:
        VO_System_Critical := TRUE;

        IF (VI_Root_Cause = E_System_Root_Cause.ROOT_GAS_LEAK OR
            VI_Root_Cause = E_System_Root_Cause.ROOT_CO_CRITICAL) AND
            VI_Freeze_Risk THEN
            VO_System_Mode := E_System_Operating_Mode.MODE_FREEZE_PROTECTION;
        ELSE
            VO_System_Mode := E_System_Operating_Mode.MODE_SAFE_STOP;
        END_IF;

        CASE VI_Root_Cause OF
            E_System_Root_Cause.ROOT_FIRE:
                VO_Status_Msg := 'АВАРИЯ: ПОЖАР';
            E_System_Root_Cause.ROOT_GAS_LEAK:
                VO_Status_Msg := 'АВАРИЯ: УТЕЧКА ГАЗА';
            E_System_Root_Cause.ROOT_CO_CRITICAL:
                VO_Status_Msg := 'АВАРИЯ: КРИТИЧЕСКИЙ CO';
            E_System_Root_Cause.ROOT_WATCHDOG_FAULT:
                VO_Status_Msg := 'АВАРИЯ: WATCHDOG';
            ELSE
                VO_Status_Msg := 'АВАРИЯ СИСТЕМЫ';
        END_CASE;
END_CASE;

          
END_FUNCTION_BLOCK

FUNCTION_BLOCK FB_State_Snapshot_Manager
  VAR_INPUT
    VI_System_Time : UDINT;
    VI_Save_Req : BOOL;
    VI_Snapshot : ST_State_Snapshot;
  END_VAR
  VAR_OUTPUT
    VO_Last_ID : UDINT;
  END_VAR
  VAR
    L_Buffer : ARRAY[0..9] OF ST_State_Snapshot;
    L_Idx : INT := 0;
  END_VAR

            IF VI_Save_Req THEN
    L_Buffer[L_Idx] := VI_Snapshot;
    L_Buffer[L_Idx].timestamp_ms := VI_System_Time;
    VO_Last_ID := VI_System_Time;
    L_Idx := (L_Idx + 1) MOD 10;
END_IF;

          
END_FUNCTION_BLOCK

FUNCTION_BLOCK FB_State_Snapshot_NVRAM
  VAR_INPUT
    VI_Command : BYTE;  (* 1=SAVE, 2=LOAD *)
    VI_Snapshot_Ptr : POINTER TO ST_State_Snapshot;
    VI_System_Time_MS : UDINT;
    VI_Operator_ID : STRING(10);
    VI_IsActivePLC : BOOL;
    VI_TwoPersonConfirmation : BOOL;
  END_VAR
  VAR_OUTPUT
    VO_Done : BOOL;
    VO_Error : UDINT;
    VO_HMI_Status_Message : STRING(200);
  END_VAR
  VAR
    L_state : BYTE;
    L_step : UDINT;
    L_temp_buffer : ARRAY[1..132] OF BYTE;
    L_byte_ptr : POINTER TO BYTE;
    L_i : UDINT;
  END_VAR
  VAR CONSTANT
    C_RECORD_SIZE : UDINT := 128;
  END_VAR

            // Исправленное копирование структуры через указатель
IF VI_Snapshot_Ptr <> 0 THEN
    L_byte_ptr := ADR(VI_Snapshot_Ptr^);
    
    CASE L_state OF
        1: // СОХРАНЕНИЕ (SAVE)
            IF L_step = 0 THEN
                // Копируем всю структуру байт за байтом в буфер NVRAM
                // Используем SIZEOF(ST_State_Snapshot), чтобы не выйти за границы структуры
                FOR L_i := 0 TO (SIZEOF(ST_State_Snapshot) - 1) DO
                    IF L_i < C_RECORD_SIZE THEN
                        L_temp_buffer[L_i + 1] := L_byte_ptr[TO_INT(L_i)];
                    END_IF;
                END_FOR;
                L_step := 1;
            END_IF;
            
        2: // ЗАГРУЗКА (LOAD)
            IF L_step = 2 THEN
                // Копируем из буфера обратно в структуру
                FOR L_i := 0 TO (SIZEOF(ST_State_Snapshot) - 1) DO
                    IF L_i < C_RECORD_SIZE THEN
                        L_byte_ptr[TO_INT(L_i)] := L_temp_buffer[L_i + 1];
                    END_IF;
                END_FOR;
                VO_Done := TRUE;
                L_state := 0;
            END_IF;
    END_CASE;
END_IF;

          
END_FUNCTION_BLOCK

FUNCTION_BLOCK FB_Supply_Ventilation_Controller
  VAR_INPUT
    VI_Fire_Alarm : BOOL;
    VI_Gas_Alarm : BOOL;
  END_VAR
  VAR_OUTPUT
    VO_Fan_Speed : BYTE;
  END_VAR

            IF VI_Fire_Alarm THEN
    VO_Fan_Speed := 0; // Остановка при пожаре
ELSIF VI_Gas_Alarm THEN
    VO_Fan_Speed := 100; // Максимум при утечке газа
ELSE
    VO_Fan_Speed := 40;
END_IF;

          
END_FUNCTION_BLOCK

FUNCTION_BLOCK FB_Trend_Analyzer
  VAR_INPUT
    VI_Value : REAL;
    VI_Threshold_Percent : REAL := 10;
    VI_System_Time_MS : UDINT;
  END_VAR
  VAR_OUTPUT
    VO_Anomaly_Detected : BOOL;
    VO_Average_7D : REAL;  (* ТЗ 12.1: Скользящее среднее 7 дней *)
    VO_Diag_Label : BOOL;  (* ТЗ 12.1: Метка "диагностика" *)
  END_VAR
  VAR
    L_History : ARRAY[1..168] OF REAL;  (* Почасовые замеры на 7 дней *)
    L_Last_Hour_Time : UDINT;
    L_Idx : INT := 1;
    L_Sum : REAL;
    L_Count : INT;
    L_i : INT;
  END_VAR

            // 1. Накопление почасовой истории (ТЗ 12.1)
IF (VI_System_Time_MS - L_Last_Hour_Time) >= 3600000 OR L_Last_Hour_Time = 0 THEN
    L_Last_Hour_Time := VI_System_Time_MS;
    L_History[L_Idx] := VI_Value;
    L_Idx := (L_Idx MOD 168) + 1;
    IF L_Count < 168 THEN L_Count := L_Count + 1; END_IF;
END_IF;

// 2. Расчет среднего за 7 дней
L_Sum := 0.0;
IF L_Count > 0 THEN
    FOR L_i := 1 TO L_Count DO L_Sum := L_Sum + L_History[L_i]; END_FOR;
    VO_Average_7D := L_Sum / TO_REAL(L_Count);
END_IF;

// 3. Детекция аномалий и метка диагностики (ТЗ 12.1)
IF VO_Average_7D > 0.0 THEN
    VO_Anomaly_Detected := (ABS(VI_Value - VO_Average_7D) / VO_Average_7D * 100.0) > VI_Threshold_Percent;
    VO_Diag_Label := VO_Anomaly_Detected; // Метка ставится при отклонении
END_IF;

          
END_FUNCTION_BLOCK

FUNCTION_BLOCK FB_TwoFactor_Auth
  VAR_INPUT
    VI_System_Time_MS : UDINT;
    VI_Start_Auth : BOOL;
    VI_RFID_Tag : STRING(20);
    VI_TOTP_Code : STRING(6);
  END_VAR
  VAR_OUTPUT
    VO_Auth_Passed : BOOL;
    VO_Auth_Failed : BOOL;
    VO_Busy : BOOL;
  END_VAR
  VAR
    L_State : BYTE;  (* 0=Idle, 1=WaitRFID, 2=WaitTOTP *)
    L_Start_Timestamp : UDINT;
  END_VAR

            CASE L_State OF
    0: 
        IF VI_Start_Auth THEN
            L_State := 1;
            L_Start_Timestamp := VI_System_Time_MS;
            VO_Busy := TRUE;
        END_IF;
    1:
        IF VI_RFID_Tag <> '' THEN
            L_State := 2;
        ELSIF (VI_System_Time_MS - L_Start_Timestamp) > 30000 THEN
            L_State := 0;
            VO_Auth_Failed := TRUE;
            VO_Busy := FALSE;
        END_IF;
    2:
        IF VI_TOTP_Code <> '' THEN
            VO_Auth_Passed := TRUE;
            L_State := 0;
            VO_Busy := FALSE;
        END_IF;
END_CASE;

          
END_FUNCTION_BLOCK

FUNCTION_BLOCK FB_User_Rule_Engine
  VAR_INPUT
    VI_Rules : ARRAY[1..10] OF ST_User_Rule;
    VI_System_State : ST_System_State_Summary;  (* Текущие значения всех датчиков *)
  END_VAR
  VAR_OUTPUT
    VO_Actions : ARRAY[1..10] OF ST_Rule_Action;
  END_VAR
  VAR
    L_i : INT;
    L_Condition_Met : BOOL;
    L_Val : REAL;
    L_Applied_Priority : ARRAY[1..100] OF BYTE;  (* Приоритет примененного действия для Target_ID *)
  END_VAR

            // Сброс приоритетов перед циклом
FOR L_i := 1 TO 100 DO L_Applied_Priority[L_i] := 0; END_FOR;

FOR L_i := 1 TO 10 DO
    IF VI_Rules[L_i].Enabled THEN
        L_Condition_Met := FALSE;
        
        // Вычисление условия (ТЗ 7.4)
        CASE VI_Rules[L_i].Condition_Type OF
            1: // Температура уличная
                L_Val := VI_System_State.Outdoor_Temp;
            2: // Температура пола (Зона 1)
                L_Val := VI_System_State.Floor_Temps[1];
            3: // CO2 (Зона 1)
                L_Val := VI_System_State.CO2[1];
            4: // Охрана
                L_Val := SEL(VI_System_State.Security_Armed, 0.0, 1.0);
        END_CASE;

        CASE VI_Rules[L_i].Condition_Op OF
            1: L_Condition_Met := (L_Val > VI_Rules[L_i].Condition_Value);
            2: L_Condition_Met := (L_Val < VI_Rules[L_i].Condition_Value);
            3: L_Condition_Met := (ABS(L_Val - VI_Rules[L_i].Condition_Value) < 0.01);
        END_CASE;

        // Выполнение действия с учетом приоритета (ТЗ 7.4)
        IF L_Condition_Met THEN
             // Проверяем, не выполнялось ли уже действие для этого Target_ID с более высоким приоритетом
             IF VI_Rules[L_i].Action_Target_ID > 0 AND VI_Rules[L_i].Action_Target_ID <= 100 THEN
                 IF VI_Rules[L_i].Priority >= L_Applied_Priority[VI_Rules[L_i].Action_Target_ID] THEN
                     VO_Actions[L_i].Active := TRUE;
                     VO_Actions[L_i].Target_ID := VI_Rules[L_i].Action_Target_ID;
                     VO_Actions[L_i].Value := VI_Rules[L_i].Action_Value;
                     L_Applied_Priority[VI_Rules[L_i].Action_Target_ID] := VI_Rules[L_i].Priority;
                 ELSE
                     VO_Actions[L_i].Active := FALSE; // Игнорируем из-за низкого приоритета
                 END_IF;
             END_IF;
        ELSE
             VO_Actions[L_i].Active := FALSE;
        END_IF;
    END_IF;
END_FOR;

          
END_FUNCTION_BLOCK

FUNCTION_BLOCK FB_Valve_Test
  VAR_INPUT
    VI_System_Time : UDINT;
    VI_Start_Test : BOOL;
    VI_Current_A : REAL;
    VI_Config : ST_Valve_Test_Config;  (* ТЗ 12.2 *)
  END_VAR
  VAR_OUTPUT
    VO_Test_Active : BOOL;
    VO_Test_Passed : BOOL;
    VO_Deviation_Percent : REAL;  (* ТЗ 12.2 *)
    VO_Error_Code : WORD;
  END_VAR
  VAR
    L_Start_Timestamp : UDINT;
    L_Peak_Current : REAL;
    L_Reaction_Time : UDINT;
  END_VAR

            IF VI_Start_Test AND NOT VO_Test_Active THEN
    VO_Test_Active := TRUE;
    L_Start_Timestamp := VI_System_Time;
    L_Peak_Current := 0.0;
    L_Reaction_Time := 0;
END_IF;

IF VO_Test_Active THEN
    IF VI_Current_A > L_Peak_Current THEN L_Peak_Current := VI_Current_A; END_IF;
    
    // Определение времени реакции (ток превысил 100мА)
    IF L_Reaction_Time = 0 AND VI_Current_A > 100.0 THEN
        L_Reaction_Time := VI_System_Time - L_Start_Timestamp;
    END_IF;

    IF (VI_System_Time - L_Start_Timestamp) > 15000 THEN
        VO_Test_Active := FALSE;
        
        // ТЗ 12.2: Контроль отклонения > 30% от номинала
        VO_Deviation_Percent := ABS(L_Peak_Current - VI_Config.Nominal_Current) / VI_Config.Nominal_Current * 100.0;
        
        VO_Test_Passed := (VO_Deviation_Percent <= 30.0) AND (L_Reaction_Time < 5000);
        
        IF NOT VO_Test_Passed THEN
            VO_Error_Code := 16#E122; // Valve Test Failed
        END_IF;
    END_IF;
END_IF;

          
END_FUNCTION_BLOCK

FUNCTION_BLOCK FB_Ventilation_System_Manager
  VAR_INPUT
    VI_System_Time_MS : UDINT;
    VI_IsActivePLC : BOOL;
    VI_CO2 : ARRAY[1..8] OF REAL;
    VI_Humidity : ARRAY[1..8] OF REAL;
    VI_Gas_Alarm : BOOL;
    VI_Fire_Alarm : BOOL;
    VI_Flood_Alarm : BOOL;
    VI_Config : ST_Ventilation_Config;
    VI_PV3_Boost : BOOL;  (* ТЗ 5.1 *)
    VI_Supply_100_Req : BOOL;  (* ТЗ 6.4 *)
    VI_Exhaust_100_Req : BOOL;  (* ТЗ 6.4 *)
    VI_Supply_80_Req : BOOL;  (* ТЗ 5.4 *)
    VI_Wet_Zone_Lights : ARRAY[1..4] OF BOOL;  (* ТЗ 4.0 *)
  END_VAR
  VAR_OUTPUT
    VO_Supply_Fans : ARRAY[1..3] OF REAL;  (* 0-100% *)
    VO_Exhaust_Fans : ARRAY[1..5] OF REAL;  (* 0-100% *)
    VO_Status : ARRAY[1..8] OF ST_Ventilation_Unit;
  END_VAR
  VAR
    L_Mode : BYTE;  (* 0-Eco, 1-Std, 2-Int, 3-Emergency *)
    L_Base_Speed : REAL;
    L_i : INT;
    L_Max_CO2 : REAL;
    L_Max_Hum : REAL;
    L_Is_Night : BOOL;
    L_Current_Time : TOD;
    L_Wet_Zone_Timers : ARRAY[1..4] OF TON;
  END_VAR

            // ========================================
// Ventilation policy layer (phase3/v2)
// ========================================
GVL_STATE.G_Ventilation_IO_Fault := FALSE;
GVL_STATE.G_Ventilation_Subsystem_Degraded := FALSE;
L_Vent_V2_Shadow_Diff_Found := FALSE;
L_Vent_V2_Switch_Enabled := TRUE;
L_Vent_V2_Path_Ready := FALSE;
L_Vent_Using_Legacy_Fallback := TRUE;
L_Policy_Normal := (VI_System_Mode = E_System_Operating_Mode.MODE_NORMAL);
L_Policy_Safe_Stop := (VI_System_Mode = E_System_Operating_Mode.MODE_SAFE_STOP);
L_Policy_Degraded := (VI_System_Mode = E_System_Operating_Mode.MODE_DEGRADED);
L_Policy_Freeze_Protection := (VI_System_Mode = E_System_Operating_Mode.MODE_FREEZE_PROTECTION);

IF NOT VI_IsActivePLC THEN
    FOR L_i := 1 TO GVL_CONSTANTS.C_MAX_SUPPLY_FANS DO
        VO_Supply_Fans[L_i] := 0;
        IF L_i <= GVL_CONSTANTS.C_MAX_SUPPLY_TEMPS THEN
            VO_Heater_Power[L_i] := 0.0;
        END_IF;
    END_FOR;
    FOR L_i := 1 TO GVL_CONSTANTS.C_MAX_EXHAUST_FANS DO
        VO_Exhaust_Fans[L_i] := 0;
    END_FOR;
    VO_Status_Msg := 'ВЕНТИЛЯЦИЯ: РЕЗЕРВНЫЙ ПЛК';
    RETURN;
END_IF;

// Проверка связи с модулями ввода-вывода
FOR L_i := 1 TO GVL_CONSTANTS.C_MAX_MODULES DO
    IF NOT VI_IO_Modules_Online[L_i] THEN
        GVL_STATE.G_Ventilation_IO_Fault := TRUE;
        // Переход в безопасное состояние при потере связи (отключение вентиляции)
        FOR L_j := 1 TO GVL_CONSTANTS.C_MAX_SUPPLY_FANS DO
            VO_Supply_Fans[L_j] := 0;
        END_FOR;
        FOR L_j := 1 TO GVL_CONSTANTS.C_MAX_EXHAUST_FANS DO
            VO_Exhaust_Fans[L_j] := 0;
        END_FOR;
        FOR L_j := 1 TO GVL_CONSTANTS.C_MAX_BOILERS DO
            VO_Heater_Power[L_j] := 0.0;
        END_FOR;
        VO_Status_Msg := 'ОШИБКА: Потеря связи с модулями ввода-вывода';
        RETURN;
    END_IF;
END_FOR;

// =========================
// SYSTEM MODE OVERRIDE
// =========================
// VENT_POLICY_ROUTING_PHASE3_V2
IF L_Policy_Safe_Stop THEN
    FOR L_i := 1 TO GVL_CONSTANTS.C_MAX_SUPPLY_FANS DO
        VO_Supply_Fans[L_i] := 0;
    END_FOR;
    FOR L_i := 1 TO GVL_CONSTANTS.C_MAX_EXHAUST_FANS DO
        VO_Exhaust_Fans[L_i] := 0;
    END_FOR;
    FOR L_i := 1 TO GVL_CONSTANTS.C_MAX_BOILERS DO
        VO_Heater_Power[L_i] := 0.0;
    END_FOR;
    VO_Status_Msg := 'ВЕНТИЛЯЦИЯ: ОСТАНОВЛЕНА POLICY SAFE_STOP';
    RETURN;
END_IF;

IF L_Policy_Degraded THEN
    FOR L_i := 1 TO GVL_CONSTANTS.C_MAX_SUPPLY_FANS DO
        VO_Supply_Fans[L_i] := 0;
    END_FOR;
    FOR L_i := 1 TO GVL_CONSTANTS.C_MAX_BOILERS DO
        VO_Heater_Power[L_i] := 0.0;
    END_FOR;
    GVL_STATE.G_Ventilation_Subsystem_Degraded := TRUE;
    VO_Status_Msg := 'ВЕНТИЛЯЦИЯ: DEGRADED POLICY';
END_IF;

IF L_Policy_Freeze_Protection THEN
    FOR L_i := 1 TO GVL_CONSTANTS.C_MAX_SUPPLY_FANS DO
        VO_Supply_Fans[L_i] := 0;
    END_FOR;
    FOR L_i := 1 TO GVL_CONSTANTS.C_MAX_EXHAUST_FANS DO
        VO_Exhaust_Fans[L_i] := 0;
    END_FOR;
    FOR L_i := 1 TO GVL_CONSTANTS.C_MAX_BOILERS DO
        VO_Heater_Power[L_i] := 0.0;
    END_FOR;
    VO_Status_Msg := 'ВЕНТИЛЯЦИЯ: FREEZE_PROTECTION POLICY (stop)';
    RETURN;
END_IF;

// MODE_FREEZE_PROTECTION пока оставляем на текущей штатной логике

// 1. Определение базовой скорости и целевой температуры по сценарию (ТЗ 7.1)
CASE VI_Current_Scenario OF
    E_SCENARIO_TYPE.SCENARIO_AWAY:
        L_Base_Speed := VI_Config.Scenario_Modes[3].Base_Fan_Speed;
        L_Target_Temp := VI_Config.Scenario_Modes[3].Target_Temp;
    E_SCENARIO_TYPE.SCENARIO_SLEEP:
        L_Base_Speed := VI_Config.Scenario_Modes[2].Base_Fan_Speed;
        L_Target_Temp := VI_Config.Scenario_Modes[2].Target_Temp;
    ELSE // PRESENCE, MORNING, EVENING
        L_Base_Speed := VI_Config.Scenario_Modes[1].Base_Fan_Speed;
        L_Target_Temp := VI_Config.Scenario_Modes[1].Target_Temp;
END_CASE;

// 2. Логика управления приточными установками (П-1, П-2, П-3)
FOR L_i := 1 TO GVL_CONSTANTS.C_MAX_SUPPLY_FANS DO
    // ПИД-регулирование мощности электрического калорифера
    IF L_i <= GVL_CONSTANTS.C_MAX_SUPPLY_TEMPS THEN
        L_PID_Heaters[L_i](
            VI_SetPoint := L_Target_Temp,
            VI_ProcessValue := VI_Supply_Temps[L_i], // Используем датчик температуры после калорифера
            VI_Kp := 4.0, VI_Tn := 120.0, VI_Tv := 0.0,
            VI_Y_Min := 0.0, VI_Y_Max := 100.0, VI_Cycle_Time_S := 1.0,
            VO_Output => VO_Heater_Power[L_i]
        );
    END_IF;

    // Определение скорости приточного вентилятора
    VO_Supply_Fans[L_i] := L_Base_Speed;
    
    // Обработка действий от Rule Engine
    FOR L_j := 1 TO GVL_CONSTANTS.C_MAX_RULES DO
        IF VI_Rule_Actions[L_j].Active AND VI_Rule_Actions[L_j].Target_ID = L_i THEN
            IF VI_Rule_Actions[L_j].Action_Type = E_Rule_Action_Type.ACTION_SET_VENTILATION THEN
                VO_Supply_Fans[L_i] := REAL_TO_BYTE(VI_Rule_Actions[L_j].Value);
            END_IF;
        END_IF;
    END_FOR;
    
    // Requests are observed but must not bypass policy directly.
    IF VI_Supply_100_Req OR VI_Supply_80_Req OR VI_Fire_Alarm OR VI_Vent_Stop OR VI_Gas_Alarm OR VI_PV3_Boost_Req THEN
        GVL_STATE.G_Ventilation_Subsystem_Degraded := TRUE;
    END_IF;
END_FOR;

// 3. Логика управления вытяжными установками (В-1 .. В-5)
FOR L_i := 1 TO GVL_CONSTANTS.C_MAX_EXHAUST_FANS DO
    VO_Exhaust_Fans[L_i] := L_Base_Speed;
    
    // ТЗ 4.0: Логика вытяжки в санузлах
    FOR L_j := 1 TO GVL_CONSTANTS.C_MAX_WET_ZONES DO
        IF VI_Config.wet_zone_to_exhaust_map[L_j] = L_i THEN
            // Включение по свету, выключение с задержкой 5 минут (используем TOF)
            L_Wet_Zone_Timers[L_j](IN := VI_Wet_Zone_Active[L_j], PT := T#5m, VI_System_Time_MS := VI_System_Time_MS);
            IF VI_Wet_Zone_Active[L_j] THEN
                VO_Exhaust_Fans[L_i] := 80; // Повышенная скорость при присутствии
            ELSIF L_Wet_Zone_Timers[L_j].Q THEN
                VO_Exhaust_Fans[L_i] := 50; // Скорость выбега (пока таймер TOF активен)
            END_IF;
        END_IF;
    END_FOR;

    // Requests are observed but must not bypass policy directly.
    IF (L_i = VI_Config.pv3_exhaust_index AND VI_PV3_Boost_Req) OR VI_Exhaust_100_Req OR VI_Fire_Alarm OR VI_Vent_Stop OR VI_Gas_Alarm THEN
        GVL_STATE.G_Ventilation_Subsystem_Degraded := TRUE;
    END_IF;
END_FOR;








// ========================================
// VENT_FINAL_CLAMP
// ========================================
IF L_Policy_Degraded THEN
    FOR L_i := 1 TO GVL_CONSTANTS.C_MAX_EXHAUST_FANS DO
        VO_Exhaust_Fans[L_i] := MIN(VO_Exhaust_Fans[L_i], VI_Config.Degraded_Exhaust_Limit);
    END_FOR;
END_IF;

// Ventilation V2 shadow runtime integration (diagnostic only)
fbVentilationV2Staging(
    VI_Zone_ID := 1,
    VI_Enable := (NOT L_Policy_Safe_Stop) AND (NOT L_Policy_Freeze_Protection) AND (NOT GVL_STATE.G_Ventilation_IO_Fault),
    VI_Fan_Speed_Setpoint := BYTE_TO_REAL(VO_Supply_Fans[1]),
    VI_Damper_Position_Setpoint := 0.0,
    VI_Heat_Recovery_Enabled := L_Policy_Normal,
    VI_Is_Active := (VO_Supply_Fans[1] > 0) OR (VO_Exhaust_Fans[1] > 0),
    VI_Fan_Speed_Actual := BYTE_TO_REAL(VO_Supply_Fans[1]),
    VI_Supply_Temp := VI_Supply_Temps[1],
    VI_Extract_Temp := VI_Room_Temps[1],
    VI_Filter_Dirty := FALSE,
    VI_Alarm_Active := GVL_STATE.G_Ventilation_IO_Fault OR GVL_STATE.G_Ventilation_Subsystem_Degraded,
    VO_Command_Shadow => L_Vent_Command_Shadow,
    VO_State_Shadow => L_Vent_State_Shadow
);

// Ventilation V2 shadow validation
IF ABS(BYTE_TO_REAL(VO_Supply_Fans[1]) - L_Vent_Command_Shadow.Fan_Speed_Setpoint) > 0.1 THEN
    L_Vent_V2_Shadow_Diff_Found := TRUE;
END_IF;
IF ABS(VI_Supply_Temps[1] - L_Vent_State_Shadow.Supply_Temp) > 0.1 THEN
    L_Vent_V2_Shadow_Diff_Found := TRUE;
END_IF;

// Guarded Ventilation V2 enable
IF L_Vent_V2_Switch_Enabled THEN
    IF NOT L_Vent_V2_Shadow_Diff_Found THEN
        L_Vent_V2_Path_Ready := TRUE;
        L_Vent_Using_Legacy_Fallback := FALSE;
    ELSE
        L_Vent_V2_Path_Ready := FALSE;
        L_Vent_Using_Legacy_Fallback := TRUE;
    END_IF;
ELSE
    L_Vent_V2_Path_Ready := FALSE;
    L_Vent_Using_Legacy_Fallback := TRUE;
END_IF;

// 4. Формирование статусного сообщения
IF L_Policy_Safe_Stop THEN
    VO_Status_Msg := 'ВЕНТИЛЯЦИЯ: ОСТАНОВЛЕНА POLICY SAFE_STOP';
ELSIF L_Policy_Freeze_Protection THEN
    VO_Status_Msg := 'ВЕНТИЛЯЦИЯ: FREEZE_PROTECTION POLICY (stop)';
ELSIF L_Policy_Degraded THEN
    VO_Status_Msg := 'ВЕНТИЛЯЦИЯ: DEGRADED POLICY';
ELSE
    VO_Status_Msg := 'Вентиляция работает в штатном режиме';
END_IF;

          
END_FUNCTION_BLOCK

FUNCTION_BLOCK FB_Water_Leakage_Manager
  VAR_INPUT
    VI_System_Time_MS : UDINT;
    VI_IsActivePLC : BOOL;
    VI_Sensors : ARRAY[1..12] OF BOOL;
    VI_Valve_35_Current : REAL;
    VI_Valve_36_Current : REAL;
    VI_Emergency_Open_Req : BYTE;  (* 1, 3, 5 мин *)
    VI_Config : ST_Flood_Config;  (* ТЗ 4.4 *)
    VI_Power_OK : BOOL;  (* ТЗ 4.3: Мониторинг питания *)
    VI_Two_Stage_Confirm : BOOL;  (* ТЗ 4.4: Подтверждение *)
  END_VAR
  VAR_OUTPUT
    VO_Valve_35_Close : BOOL;
    VO_Valve_36_Close : BOOL;
    VO_Flood_Alarm : BOOL;
    VO_Alert_Priority : BYTE;  (* ТЗ 4.3: 1-Low, 2-Normal, 3-Critical *)
    VO_Status_Msg : STRING(200);
  END_VAR
  VAR
    L_Zone1_Alarm : BOOL;
    L_Zone2_Alarm : BOOL;
    L_Zone3_Alarm : BOOL;
    L_Emergency_Timer : TON;
    L_Confirm_Timer : TON;
    L_Confirm_Wait : BOOL;
    L_Emergency_Count : UINT;  (* ТЗ 4.4: Лимит 3 раза в сутки *)
    L_Day_Timer : TON;
    L_Last_Req : BYTE;
    L_Valve_35_Error : BOOL;  (* ТЗ 4.3: Диагностика тока *)
    L_Valve_36_Error : BOOL;
  END_VAR

            IF NOT VI_IsActivePLC THEN RETURN; END_IF;

L_Any_Leak := FALSE;
L_Any_Warning := FALSE;

FOR L_i := 1 TO GVL_CONSTANTS.C_MAX_FLOOD_SENSORS DO
    L_Sensor_Timers[L_i](
        IN := VI_Sensors[L_i],
        PT := TO_TIME(VI_Config.min_duration_ms + VI_Config.warning_duration_ms),
        VI_System_Time_MS := VI_System_Time_MS
    );

    IF L_Sensor_Timers[L_i].ET >= TO_TIME(VI_Config.min_duration_ms) THEN
        L_Any_Warning := TRUE;

        IF L_Sensor_Timers[L_i].Q THEN
            L_Any_Leak := TRUE;

            IF VI_Config.sensor_to_valve_map[L_i] = 1 THEN
                VO_Close_Valve_35 := TRUE;
            ELSIF VI_Config.sensor_to_valve_map[L_i] = 2 THEN
                VO_Close_Valve_36 := TRUE;
            END_IF;
        END_IF;
    END_IF;
END_FOR;

// Health signals
VO_Leak_Detected := L_Any_Leak;
VO_Leak_Warning_Level := L_Any_Warning;

// Status
IF L_Any_Leak THEN
    VO_Status_Msg := 'АВАРИЯ: ПРОТЕЧКА ВОДЫ. КЛАПАНЫ ЗАКРЫТЫ.';
ELSIF L_Any_Warning THEN
    VO_Status_Msg := 'ПРЕДУПРЕЖДЕНИЕ: ОБНАРУЖЕНА ВОДА.';
ELSE
    VO_Status_Msg := 'Система контроля протечек в норме';
    VO_Close_Valve_35 := FALSE;
    VO_Close_Valve_36 := FALSE;
END_IF;

          
END_FUNCTION_BLOCK

FUNCTION_BLOCK FB_Water_Valve_Controller IMPLEMENTS IValveController
  VAR_INPUT
    VI_IsActivePLC : BOOL;
    VI_Valve_Type : E_VALVE_TYPE;
    VI_Current_Feedback : REAL;  (* Ток двигателя *)
    VI_Limit_Open : BOOL;  (* Концевик открыто *)
    VI_Limit_Closed : BOOL;  (* Концевик закрыто *)
    VI_System_Time : UDINT;
  END_VAR
  VAR_OUTPUT
    VO_Valve_Open_Cmd : BOOL;
    VO_Valve_Close_Cmd : BOOL;
    VO_Status : BYTE;  (* 0-Open, 1-Closed, 2-Moving, 3-Error *)
  END_VAR
  VAR
    L_Moving : BOOL;
    L_Move_Start_Time : UDINT;
    L_Target_State : BOOL;  (* FALSE-Open, TRUE-Close *)
  END_VAR

            // Логика диагностики (п. 4.3 ТЗ)
IF L_Moving THEN
    IF (VI_System_Time - L_Move_Start_Time) > 10000 THEN // Таймаут 10 сек
        VO_Status := 3; // Ошибка
        L_Moving := FALSE;
    ELSIF (L_Target_State = TRUE AND VI_Limit_Closed) OR (L_Target_State = FALSE AND VI_Limit_Open) THEN
        VO_Status := SEL(L_Target_State, 0, 1);
        L_Moving := FALSE;
    ELSE
        VO_Status := 2; // Moving
    END_IF;
END_IF;

          

METHOD OpenValve : BOOL
  VAR_INPUT
    VI_Operator_ID : STRING(10);
    VI_Force : BOOL;
  END_VAR
                  IF VI_IsActivePLC OR VI_Force THEN
    VO_Valve_Open_Cmd := TRUE;
    VO_Valve_Close_Cmd := FALSE;
    L_Moving := TRUE;
    L_Target_State := FALSE;
    L_Move_Start_Time := VI_System_Time;
    OpenValve := TRUE;
ELSE
    OpenValve := FALSE;
END_IF;
                
END_METHOD

METHOD CloseValve : BOOL
  VAR_INPUT
    VI_Operator_ID : STRING(10);
    VI_Force : BOOL;
  END_VAR
                  IF VI_IsActivePLC OR VI_Force THEN
    VO_Valve_Open_Cmd := FALSE;
    VO_Valve_Close_Cmd := TRUE;
    L_Moving := TRUE;
    L_Target_State := TRUE;
    L_Move_Start_Time := VI_System_Time;
    CloseValve := TRUE;
ELSE
    CloseValve := FALSE;
END_IF;
                
END_METHOD

METHOD GetStatus : BYTE
                  GetStatus := VO_Status;
                
END_METHOD
END_FUNCTION_BLOCK

FUNCTION_BLOCK FB_Zone_Access_Manager
  VAR_INPUT
    VI_Operator_ID : STRING(10);
    VI_Zone_ID : BYTE;
    VI_Req_Level : BYTE;
  END_VAR
  VAR
    L_Rights : ARRAY[1..10] OF ST_Operator_Zone_Rights;
  END_VAR

            
          

METHOD CheckAccess : BOOL
  VAR_INPUT
    VI_Op : STRING(10);
    VI_Req_Level : BYTE;
  END_VAR
                  IF VI_Op = 'ADMIN' THEN
    // Если 2FA включена, проверяем флаг прохождения второго фактора
    IF GVL_HMI_Config.G_HMI_Admin_2FA_Enabled THEN
        CheckAccess := GVL_HMI_Config.G_HMI_Current_Operator_Factor2_Done;
    ELSE
        CheckAccess := TRUE;
    END_IF;
ELSIF VI_Op = 'SERVICE' AND VI_Req_Level <= 3 THEN
    CheckAccess := TRUE;
ELSE
    CheckAccess := FALSE;
END_IF;
                
END_METHOD
END_FUNCTION_BLOCK

PROGRAM PRG_Main
  VAR
    fbHeating : FB_Heating_System_Manager;  (* Менеджеры систем *)
    fbSecurity : FB_Security_System_Manager;
    fbWater : FB_Water_Leakage_Manager;
    fbGasSmoke : FB_Gas_Smoke_Manager;
    fbVentilation : FB_Ventilation_System_Manager;
    fbRuleEngine : FB_User_Rule_Engine;
    fbLightingBlinds : FB_Lighting_Blinds_Manager;
    fbSimulation : FB_Simulation_Manager;
    fbDHW : FB_DHW_Manager;  (* ТЗ 5.0 *)
    fbAccessControl : FB_Access_Control;
    fbHeartbeat : FB_PLC_Heartbeat;  (* Системные блоки *)
    fbNVRAM : FB_NVRAM_Manager;
    fbGateway : FB_Gateway_Interface;
    fbLogger : FB_Debug_Logger;
    L_Is_Active : BOOL;  (* Локальные переменные *)
    L_First_Cycle : BOOL := TRUE;
    L_System_State : ST_System_State_Summary;
    L_i : INT;
    L_Methane_LEL_Real : ARRAY[1..2] OF REAL;
    L_Manifold_Temps_Supply_Real : ARRAY[1..5] OF REAL;
    L_Manifold_Temps_Return_Real : ARRAY[1..5] OF REAL;
    L_Manifold_Pressures_Real : ARRAY[1..5] OF REAL;
    L_Manifold_Currents_Real : ARRAY[1..5] OF REAL;
    L_Current_TOD : TOD;
    L_Opening_Sensors : ARRAY[1..15] OF BOOL;  (* ТЗ 8.2: Распределение датчиков *)
    L_GlassBreak_Sensors : ARRAY[1..15] OF BOOL;
    L_Flood_Sensors : ARRAY[1..12] OF BOOL;
    L_Backup_Day : INT := 1;  (* ТЗ 16.2: Ротация 7 копий *)
  END_VAR

            // 0. Обновление системного времени
GVL_Vars.G_System_Time_MS := GVL_Vars.G_System_Time_MS + 10; 

// 1. Логика резервирования (ТЗ 11.1)
fbHeartbeat(
    VI_Local_ID := GVL_Vars.G_Local_PLC_ID,
    VI_System_Time := GVL_Vars.G_System_Time_MS,
    VI_Remote_Pulse := GVL_Vars.G_Remote_PLC_Pulse,
    VO_Is_Active => L_Is_Active
);
GVL_Vars.G_Active_PLC_ID := SEL(L_Is_Active, 0, GVL_Vars.G_Local_PLC_ID);

// 2. Инициализация и Бэкап (ТЗ 16.2)
L_Current_TOD := UDINT_TO_TOD(GVL_Vars.G_System_Time_MS MOD 86400000);
IF L_First_Cycle THEN
    L_First_Cycle := FALSE;
    fbNVRAM(VI_Command := 2, VI_RecordIndex := 1, VI_DataPtr := ADR(GVL_Vars.G_HMI_Gas_Config), VI_DataSize := SIZEOF(GVL_Vars.G_HMI_Gas_Config));
END_IF;

// Ежесуточный бэкап в 03:00 (ТЗ 16.2: Ротация 7 копий)
IF L_Current_TOD >= TOD#03:00 AND L_Current_TOD <= TOD#03:00:01 THEN
    fbNVRAM(VI_Command := 1, VI_RecordIndex := L_Backup_Day, VI_DataPtr := ADR(GVL_Vars.G_HMI_Gas_Config), VI_DataSize := SIZEOF(GVL_Vars.G_HMI_Gas_Config));
    L_Backup_Day := (L_Backup_Day MOD 7) + 1;
END_IF;

// 3. ТЗ 8.2: Параллельная обработка датчиков
FOR L_i := 1 TO 2 DO 
    L_Methane_LEL_Real[L_i] := GVL_IO.AI_Methane_LEL[L_i].rValue; 
END_FOR;
FOR L_i := 1 TO 5 DO 
    L_Manifold_Temps_Supply_Real[L_i] := GVL_IO.AI_Manifold_Temps_Supply[L_i].rValue; 
    L_Manifold_Temps_Return_Real[L_i] := TO_REAL(GVL_IO.AI_Manifold_Temps_Return[L_i]) / 10.0;
    L_Manifold_Pressures_Real[L_i] := TO_REAL(GVL_IO.AI_Manifold_Pressures[L_i]) / 100.0; // 0-10V -> 0-10.0 bar
    L_Manifold_Currents_Real[L_i] := TO_REAL(GVL_IO.AI_Manifold_Currents[L_i]) / 100.0; // 4-20mA -> 4.0-20.0 mA
END_FOR;

FOR L_i := 1 TO 15 DO
    // ПЛК A (ID=1) обрабатывает нечетные, ПЛК B (ID=2) - четные
    IF (GVL_Vars.G_Local_PLC_ID = 1 AND (L_i MOD 2 <> 0)) OR (GVL_Vars.G_Local_PLC_ID = 2 AND (L_i MOD 2 = 0)) THEN
        L_Opening_Sensors[L_i] := GVL_IO.DI_Security_Open[L_i];
        L_GlassBreak_Sensors[L_i] := GVL_IO.DI_Security_Glass[L_i];
    END_IF;
END_FOR;

FOR L_i := 1 TO 12 DO
    IF (GVL_Vars.G_Local_PLC_ID = 1 AND (L_i MOD 2 <> 0)) OR (GVL_Vars.G_Local_PLC_ID = 2 AND (L_i MOD 2 = 0)) THEN
        L_Flood_Sensors[L_i] := GVL_IO.DI_Flood_Sensors[L_i];
    END_IF;
END_FOR;

    // 4. Сбор состояния
    L_System_State.Outdoor_Temp := GVL_IO.AI_Temp_Outdoor.rValue;
    FOR L_i := 1 TO 16 DO 
        L_System_State.Floor_Temps[L_i] := GVL_IO.AI_Floor_Temps[L_i]; 
        L_System_State.Indoor_Temp[L_i] := GVL_IO.AI_Room_Temps[L_i];
        L_System_State.CO2[MIN(L_i, 8)] := 400.0; 
        L_System_State.Humidity[MIN(L_i, 8)] := 45.0; 
    END_FOR;
    L_System_State.Security_Armed := GVL_Vars.G_Security_Armed;
    L_System_State.Flood_Alarm := GVL_Vars.G_Flood_Alarm_Active;
    L_System_State.Gas_Alarm := GVL_Vars.G_Gas_Alarm_Active;
    L_System_State.Fire_Alarm := GVL_Vars.G_Fire_Alarm_Active;

    // 5. Выполнение системной логики
    fbGasSmoke(
        VI_System_Time_MS := GVL_Vars.G_System_Time_MS,
        VI_IsActivePLC := L_Is_Active,
        VI_Methane_LEL := L_Methane_LEL_Real,
        VI_CO_PPM := GVL_IO.AI_CO_PPM,
        VI_Smoke_Sensors := GVL_IO.DI_Smoke_Sensors,
        VI_Mute_Request := GVL_Vars.G_HMI_Mute_Alarm,
        VO_Gas_Alarm => GVL_Vars.G_Gas_Alarm_Active,
        VO_Fire_Alarm => GVL_Vars.G_Fire_Alarm_Active,
        VO_Gas_Valve_Close => GVL_IO.DO_Gas_Valve_Close
    );

    // ТЗ 3.6: При тревоге -> долгосрочный отъезд
    IF fbSecurity.VO_Long_Away_Req THEN
        GVL_Vars.G_Current_Scenario := E_SCENARIO_TYPE.SCENARIO_AWAY;
    END_IF;

    fbWater(
        VI_System_Time_MS := GVL_Vars.G_System_Time_MS,
        VI_IsActivePLC := L_Is_Active,
        VI_Sensors := L_Flood_Sensors,
        VI_Valve_35_Current := GVL_IO.AI_Water_Valve_35_Current,
        VI_Valve_36_Current := GVL_IO.AI_Water_Valve_36_Current,
        VI_Config := GVL_Vars.G_Flood_Config,
        VI_Power_OK := GVL_IO.DI_Power_OK,
        VO_Flood_Alarm => GVL_Vars.G_Flood_Alarm_Active,
        VO_Valve_35_Close => GVL_IO.DO_Water_Valve_35_Close,
        VO_Valve_36_Close => GVL_IO.DO_Water_Valve_36_Close
    );

    fbHeating(
        VI_System_Time_MS := GVL_Vars.G_System_Time_MS,
        VI_IsActivePLC := L_Is_Active AND NOT fbGasSmoke.VO_Boiler_Stop,
        VI_Outdoor_Temp := L_System_State.Outdoor_Temp,
        VI_Floor_Temps := GVL_IO.AI_Floor_Temps,
        VI_Room_Temps := GVL_IO.AI_Room_Temps,
        VI_Config := GVL_Vars.G_Heating_Config,
        VI_Manifold_Temps_Supply := L_Manifold_Temps_Supply_Real,
        VI_Manifold_Temps_Return := L_Manifold_Temps_Return_Real,
        VI_Manifold_Pressures := L_Manifold_Pressures_Real,
        VI_Manifold_Currents := L_Manifold_Currents_Real,
        VI_Boiler_Flame_Status := GVL_IO.AI_Boiler_Flame_Status,
        VI_Maintenance_Zones := GVL_Vars.G_Maintenance_Zones,
        VI_Maintenance_Manifolds := GVL_Vars.G_Maintenance_Manifolds,
        VO_Manifold_Pumps => GVL_IO.DO_Manifold_Pumps,
        VO_Zone_Valves => GVL_IO.DO_Zone_Valves,
        VO_Boiler_Enable => GVL_IO.DO_Boiler_Enable
    );
    // Конверсия выходов для Modbus
    FOR L_i := 1 TO 5 DO GVL_IO.AO_Manifold_Valves[L_i] := TO_UINT(fbHeating.VO_Manifold_Valves[L_i] * 10.0); END_FOR;
    FOR L_i := 1 TO 2 DO GVL_IO.AO_Boiler_Setpoint[L_i] := TO_UINT(fbHeating.VO_Boiler_Setpoint[L_i] * 10.0); END_FOR;

fbSecurity(
    VI_System_Time_MS := GVL_Vars.G_System_Time_MS,
    VI_IsActivePLC := L_Is_Active,
    VI_Opening_Sensors := L_Opening_Sensors,
    VI_GlassBreak_Sensors := L_GlassBreak_Sensors,
    VI_Config := GVL_Vars.G_Security_Config,
    VI_Group_2F_Open := GVL_IO.DI_Security_2F_Group, // ТЗ 3.1
    VI_Group_2F_Glass := GVL_IO.DI_Security_2F_Group, // ТЗ 3.2 (используем тот же канал если не выделен)
    VO_Armed => GVL_Vars.G_Security_Armed
);

fbAccessControl(
    VI_System_Time_MS := GVL_Vars.G_System_Time_MS,
    VI_IsActivePLC := L_Is_Active,
    VI_Armed := GVL_Vars.G_Security_Armed,
    VI_Gate_Open_Req := GVL_Vars.G_HMI_Gate_Open_Req,
    VI_Wicket_Open_Req := GVL_Vars.G_HMI_Wicket_Open_Req,
    VI_Lock_1_Open_Req := GVL_Vars.G_HMI_Lock_1_Open_Req,
    VI_Lock_1_Close_Req := GVL_Vars.G_HMI_Lock_1_Close_Req,
    VI_Lock_2_Open_Req := GVL_Vars.G_HMI_Lock_2_Open_Req,
    VI_Lock_2_Close_Req := GVL_Vars.G_HMI_Lock_2_Close_Req,
    VI_Config := GVL_Vars.G_Security_Config
);

// Сброс команд HMI (импульсные кнопки)
IF GVL_Vars.G_HMI_Gate_Open_Req AND NOT fbAccessControl.VO_Gate_Open THEN GVL_Vars.G_HMI_Gate_Open_Req := FALSE; END_IF;
IF GVL_Vars.G_HMI_Wicket_Open_Req AND NOT fbAccessControl.VO_Wicket_Open THEN GVL_Vars.G_HMI_Wicket_Open_Req := FALSE; END_IF;
IF GVL_Vars.G_HMI_Lock_1_Open_Req AND NOT fbAccessControl.VO_Lock_1_Open THEN GVL_Vars.G_HMI_Lock_1_Open_Req := FALSE; END_IF;
IF GVL_Vars.G_HMI_Lock_1_Close_Req AND NOT fbAccessControl.VO_Lock_1_Close THEN GVL_Vars.G_HMI_Lock_1_Close_Req := FALSE; END_IF;
IF GVL_Vars.G_HMI_Lock_2_Open_Req AND NOT fbAccessControl.VO_Lock_2_Open THEN GVL_Vars.G_HMI_Lock_2_Open_Req := FALSE; END_IF;
IF GVL_Vars.G_HMI_Lock_2_Close_Req AND NOT fbAccessControl.VO_Lock_2_Close THEN GVL_Vars.G_HMI_Lock_2_Close_Req := FALSE; END_IF;

// Маппинг на физические выходы
GVL_IO.DO_Gate_Open := fbAccessControl.VO_Gate_Open;
GVL_IO.DO_Wicket_Open := fbAccessControl.VO_Wicket_Open;
GVL_IO.DO_Lock_1_Open := fbAccessControl.VO_Lock_1_Open;
GVL_IO.DO_Lock_1_Close := fbAccessControl.VO_Lock_1_Close;
GVL_IO.DO_Lock_2_Open := fbAccessControl.VO_Lock_2_Open;
GVL_IO.DO_Lock_2_Close := fbAccessControl.VO_Lock_2_Close;

fbDHW(
    VI_System_Time_MS := GVL_Vars.G_System_Time_MS,
    VI_IsActivePLC := L_Is_Active,
    VI_Temp := GVL_IO.AI_DHW_Temp,
    VI_Pressure := GVL_IO.AI_DHW_Pressure,
    VI_Config := GVL_Vars.G_DHW_Config,
    VI_Maintenance := GVL_Vars.G_Maintenance_Lighting[1] // Условно используем ячейку для ГВС
);
GVL_IO.DO_DHW_Heating_Pump := fbDHW.VO_Heating_Pump;
GVL_IO.DO_DHW_Circ_Pump := fbDHW.VO_Circ_Pump;

fbVentilation(
    VI_System_Time_MS := GVL_Vars.G_System_Time_MS,
    VI_IsActivePLC := L_Is_Active,
    VI_CO2 := L_System_State.CO2,
    VI_Humidity := L_System_State.Humidity,
    VI_Gas_Alarm := GVL_Vars.G_Gas_Alarm_Active,
    VI_Fire_Alarm := GVL_Vars.G_Fire_Alarm_Active,
    VI_Flood_Alarm := GVL_Vars.G_Flood_Alarm_Active,
    VI_Config := GVL_Vars.G_Ventilation_Config,
    VI_PV3_Boost := fbGasSmoke.VO_Vent_PV3_Boost, // ТЗ 5.1
    VI_Supply_100_Req := fbGasSmoke.VO_Supply_100_Req, // ТЗ 6.4
    VI_Exhaust_100_Req := fbGasSmoke.VO_Exhaust_100_Req, // ТЗ 6.4
    VI_Supply_80_Req := fbGasSmoke.VO_Supply_80_Req, // ТЗ 5.4
    VI_Wet_Zone_Lights := fbLightingBlinds.VO_Wet_Zone_Light_Active // ТЗ 4.0
);
// Конверсия выходов вентиляции
FOR L_i := 1 TO 3 DO GVL_IO.AO_Supply_Fans[L_i] := TO_UINT(fbVentilation.VO_Supply_Fans[L_i] * 10.0); END_FOR;
FOR L_i := 1 TO 5 DO GVL_IO.AO_Exhaust_Fans[L_i] := TO_UINT(fbVentilation.VO_Exhaust_Fans[L_i] * 10.0); END_FOR;

fbSimulation(
    VI_System_Time_MS := GVL_Vars.G_System_Time_MS,
    VI_Enabled := (GVL_Vars.G_Current_Scenario = E_SCENARIO_TYPE.SCENARIO_AWAY),
    VI_Intensity := 0.3
);

fbLightingBlinds(
    VI_System_Time_MS := GVL_Vars.G_System_Time_MS,
    VI_IsActivePLC := L_Is_Active,
    VI_Current_Scenario := GVL_Vars.G_Current_Scenario,
    VI_Away_Level := fbSecurity.VO_Away_Level,
    VI_Simulation_Active := (GVL_Vars.G_Current_Scenario = E_SCENARIO_TYPE.SCENARIO_AWAY),
    VI_Simulation_Lights := fbSimulation.VO_Light_States,
    VI_Physical_Switches := GVL_IO.DI_Lighting_Switches, // ТЗ 1.0
    VI_Motion_Sensors := GVL_IO.DI_Motion_Sensors, // ТЗ 2.0
    VI_Maintenance := GVL_Vars.G_Maintenance_Lighting // ТЗ 6.0
);

fbRuleEngine(VI_System_State := L_System_State);

fbGateway(
    VI_System_Time_MS := GVL_Vars.G_System_Time_MS,
    VI_Local_PLC_Role := SEL(L_Is_Active, E_PLC_ROLE.ROLE_STANDBY, E_PLC_ROLE.ROLE_ACTIVE),
    VI_FloorHeating_Temps := GVL_IO.AI_Floor_Temps,
    VI_Room_Temps := GVL_IO.AI_Room_Temps,
    VI_Zone_Valve_States := GVL_IO.DO_Zone_Valves,
    VI_Manifold_Pressures := L_Manifold_Pressures_Real,
    VI_Manifold_Pump_States := GVL_IO.DO_Manifold_Pumps,
    VI_Outdoor_Temp := L_System_State.Outdoor_Temp,
    VI_Security_Armed := GVL_Vars.G_Security_Armed,
    VI_Flood_Alarm_Active := GVL_Vars.G_Flood_Alarm_Active,
    VI_Gas_Alarm_Active := GVL_Vars.G_Gas_Alarm_Active,
    VI_Fire_Alarm_Active := GVL_Vars.G_Fire_Alarm_Active,
    VI_Lighting_Base_Levels := fbLightingBlinds.VO_Lighting_Levels,
    VI_Blinds_Positions := fbLightingBlinds.VO_Blinds_Positions,
    VI_Active_Scenario := GVL_Vars.G_Current_Scenario
);

          
END_PROGRAM
